ACTION Robi_PallWait_action:
Robot01.PosNo:=POS_FEED_PAL_WAIT;
	Robot01.PosOffset:=gRobotOffset;
	Robot01.Override:=MP.ST00.Override;
	Robot01.SetToolOn:=FALSE;
	Robot01.SetToolOff:=TRUE;
	Robot01.ExecuteMove:=TRUE;
END_ACTION

ACTION Release_Nest_2_action:
ST00_71_K2.SetSignalHigh:=TRUE; (* Schnittstelle Bedrucken Tinte Abholposition frei *)
END_ACTION

ACTION ST08_Pallett_5_entry:
ProcessMessage01:='';
END_ACTION

ACTION ST08_Pallett_5_action:
ProcessMessage01:='1IM7';(*warte Pallette*)
END_ACTION

ACTION ST08_Pallett_5_exit:
ST08_Process.Start:=FALSE;
ProcessMessage01:='';
END_ACTION

ACTION Robot01_PosPal_5_entry:
IF 	PosIdx<TD.PartsInRoboGripper THEN
	PosIdx:=TD.PartsInRoboGripper;
END_IF

(*für das ausschleusen der Testteile mit einem Blister*)
IF	(gTakeTestParts OR gTakeTestPartsAuto) AND
	PosIdx <= MP.ST03.NoOfTestParts THEN
	CTR:=PosIdx;
END_IF
END_ACTION

ACTION Robot01_PosPal_5_action:
Robot01.PosNo:=POS_FEED_PAL_WAIT + (PosIdx/TD.PartsInRoboGripper);
Robot01.PosOffset:=gRobotOffset;
Robot01.Override:=MP.ST00.Override;
Robot01.SetToolOn:=TRUE;
Robot01.SetToolOff:=FALSE;
Robot01.ExecuteMove:=TRUE;
END_ACTION

ACTION Robot01_PosPal_5_exit:
gRob01GripState:=PART_NO;
PosIdx:=PosIdx+ TD.PartsInRoboGripper;
gPartsInserted:=gPartsInserted+ TD.PartsInRoboGripper;
gPartsTest:=gPartsTest+ TD.PartsInRoboGripper;
END_ACTION

ACTION Reset_Test2_action:
(*für das ausschleusen der Testteile mit einem Blister*)
IF	(gTakeTestParts OR gTakeTestPartsAuto) AND
	CTR>= MP.ST03.NoOfTestParts THEN
	ST08_Palletizing.TestpartMoveOut:=TRUE;
	CTR:=0;
	gTakeTestParts:=FALSE;
	gTakeTestPartsAuto:=FALSE;
	TestPartsRemove := TRUE;
END_IF
END_ACTION

ACTION Release_Nest_21_action:
ST00_71_K2.SetSignalHigh:=TRUE; (* Schnittstelle Bedrucken Tinte Abholposition frei *)
END_ACTION

ACTION ST08_Pallett_51_action:
IF ST08_Process.State=STATE_WAIT THEN
	ST08_Process.Start:=TRUE;
END_IF
END_ACTION

ACTION Robot01_Pos51_action:
Robot01.PosNo:=POS_NOK;
Robot01.PosOffset:=gRobotOffset;
Robot01.Override:=MP.ST00.Override;
Robot01.SetToolOn:=TRUE;
Robot01.SetToolOff:=FALSE;
Robot01.ExecuteMove:=TRUE;
END_ACTION

ACTION Robot01_TestPos__entry:
CTR:=CTR+1;
END_ACTION

ACTION Robot01_TestPos__action:
Robot01.PosNo:=POS_TEST_PARTS ;
Robot01.PosOffset:=gRobotOffset;
Robot01.Override:=MP.ST00.Override;
Robot01.SetToolOn:=TRUE;
Robot01.SetToolOff:=FALSE;
Robot01.ExecuteMove:=TRUE;
END_ACTION

ACTION Robot01_TestPos__exit:
gRob01GripState:=PART_NO;
END_ACTION

ACTION Reset_Test__action:
IF CTR>=MP.ST03.NoOfTestParts THEN
	CTR:=0;
	gTakeTestParts:=FALSE;
	gTakeTestPartsAuto:=FALSE;
	TestPartsRemove:=TRUE;
END_IF
END_ACTION

ACTION Robot01_POS_PARK_12_action:
Robot01.PosNo:=POS_PARK;
Robot01.PosOffset:=gRobotOffset;
Robot01.Override:=MP.ST00.Override;
Robot01.SetToolOn:=FALSE;
Robot01.SetToolOff:=FALSE;
Robot01.ExecuteMove:=TRUE;
END_ACTION

ACTION Close_Stopper____________action:
ST03_422_Y64_6.MoveInit:=TRUE;
END_ACTION

ACTION Open_Seperator__________action:
ST03_422_Y64_5.MoveInit:=TRUE;	(* Förderband  Stopper Vereinzler AST/GST *)
END_ACTION

ACTION Wait__for_Part_____entry:
ProcessMessage01:='';
Delay.IN:=FALSE;
Delay();
END_ACTION

ACTION Wait__for_Part_____action:
ProcessMessage01:='1IM6';(*warte auf Teil in Vereinzelung*)
Delay.IN:= ST03_421_B63_7.BitInToCheck; 			 (* Schnittstelle Iso auf Übergabeposition *)
Delay.PT:=T#500ms;
Delay();
END_ACTION

ACTION Wait__for_Part_____exit:
ProcessMessage01:='';
END_ACTION

ACTION Close__seperator__action:
ST03_422_Y64_5.MoveWork:=TRUE;
END_ACTION

ACTION Open__Stopper___action:
ST03_422_Y64_6.MoveWork:=TRUE;
END_ACTION

ACTION Wait_for__Part___entry:
ProcessMessage01:='';
Delay.IN:=FALSE;
Delay();
END_ACTION

ACTION Wait_for__Part___action:
ProcessMessage01:='1IM10';(*warte auf Teil in Abholpositon*)
Delay.IN:=ST03_422_B64_4.BitInToCheck; 		 (* Teil auf Abholposition Roboter *)
Delay.PT:=T#500ms;
Delay();
END_ACTION

ACTION Wait_for__Part___exit:
ProcessMessage01:='';
END_ACTION

ACTION Close_Stopper_2___________action:
ST03_422_Y64_6.MoveInit:=TRUE;
END_ACTION

ACTION Open_Seperator_2_________action:
ST03_422_Y64_5.MoveInit:=TRUE;	(* Förderband  Stopper Vereinzler AST/GST *)
END_ACTION

ACTION Close_Stopper__action:
ST08_412_Y55_2.MoveWork:=TRUE;
END_ACTION

ACTION Open_seperator__action:
ST08_412_Y55_0.MoveInit:=TRUE;
END_ACTION

ACTION Wait_for_Part__entry:
ProcessMessage01:='';
Delay.IN:=FALSE;
Delay();
END_ACTION

ACTION Wait_for_Part__action:
ProcessMessage01:='1IM6';(*warte auf Teil in Vereinzelung*)
Delay.IN:=ST08_412_B58_7.BitInToCheck; 		 (* Schnittstelle Iso auf Übergabeposition *)
Delay.PT:=T#50ms;
Delay();
END_ACTION

ACTION Wait_for_Part__exit:
ProcessMessage01:='';
END_ACTION

ACTION Move_Dist_entry:
IstPosHelp:=ST03_51_M1.sPos.ist;
END_ACTION

ACTION Close_seperator__action:
ST08_412_Y55_0.MoveWork:=TRUE;
END_ACTION

ACTION Open_Stopper___action:
ST08_412_Y55_2.MoveInit:=TRUE;
END_ACTION

ACTION Wait_for_Part___entry:
ProcessMessage01:='';
Delay.IN:=FALSE;
Delay();
END_ACTION

ACTION Wait_for_Part___action:
ProcessMessage01:='1IM10';(*warte auf Teil in Abholpositon*)
Delay.IN:=ST08_412_B59_0.BitInToCheck; 		 (* Teil auf Abholposition Roboter *)
Delay.PT:=T#500ms;
Delay();
END_ACTION

ACTION Wait_for_Part___exit:
ProcessMessage01:='';
END_ACTION

ACTION Close_Stopper_______action:
ST08_412_Y55_2.MoveWork:=TRUE;
END_ACTION

ACTION Open_seperator_______action:
ST08_412_Y55_0.MoveInit:=TRUE;
END_ACTION

ACTION Robot01_Pos35_action:
Robot01.PosNo:=POS_WT_POS2;
Robot01.PosOffset:=gRobotOffset;
Robot01.Override:=MP.ST00.Override;
Robot01.SetToolOn:=FALSE;
Robot01.SetToolOff:=TRUE;
Robot01.ExecuteMove:=TRUE;
END_ACTION

ACTION Robot01_Pos35_exit:
gRob01GripState:=PART_OK;
END_ACTION

ACTION Stopp_Band_91pol_action:
(* Bei 91 poligen Stecker das Band anhalten*)

IF 	gTypeCode=379 THEN
	ST03_51_M1.MotorOn:=FALSE;
	ST03_51_M1.MotorOff :=TRUE;
END_IF
END_ACTION

ACTION Robot01_Pos31_65_action:
Robot01.PosNo:=POS_WT_POS1;
Robot01.PosOffset:=gRobotOffset;
Robot01.Override:=MP.ST00.Override;
Robot01.SetToolOn:=FALSE;
Robot01.SetToolOff:=TRUE;
Robot01.ExecuteMove:=TRUE;
END_ACTION

ACTION Robot01_Pos31_65_exit:
gRob01GripState:=PART_OK;
END_ACTION

ACTION Band_starten_action:
(* Band wieder starten*)

IF 	gTypeCode=379 THEN
	ST03_51_M1.MotorOn:=TRUE;
	ST03_51_M1.MotorOff :=FALSE;
END_IF
END_ACTION

ACTION Robot01__POS_PARK_action:
Robot01.PosNo:=POS_PARK;
Robot01.PosOffset:=gRobotOffset;
Robot01.Override:=MP.ST00.Override;
Robot01.SetToolOn:=FALSE;
Robot01.SetToolOff:=FALSE;
Robot01.ExecuteMove:=TRUE;
END_ACTION

ACTION ST08_Pallett_6_entry:
ProcessMessage01:='';
END_ACTION

ACTION ST08_Pallett_6_action:
ProcessMessage01:='1IM7';(*warte Pallette*)
END_ACTION

ACTION ST08_Pallett_6_exit:
ST08_Process.Start:=FALSE;
ProcessMessage01:='';
END_ACTION

ACTION Robot01_PosPal_65_entry:
IF 	PosIdx<TD.PartsInRoboGripper THEN
	PosIdx:=TD.PartsInRoboGripper;
END_IF

(*für das ausschleusen der Testteile mit einem Blister*)
IF	(gTakeTestParts OR gTakeTestPartsAuto) AND
	PosIdx <= MP.ST03.NoOfTestParts THEN
	CTR:=PosIdx;
END_IF
END_ACTION

ACTION Robot01_PosPal_65_action:
Robot01.PosNo:=POS_FEED_PAL_WAIT + PosIdx;
Robot01.PosOffset:=gRobotOffset;
Robot01.Override:=MP.ST00.Override;
Robot01.SetToolOn:=TRUE;
Robot01.SetToolOff:=FALSE;
Robot01.ExecuteMove:=TRUE;
END_ACTION

ACTION Robot01_PosPal_65_exit:
gRob01GripState:=PART_NO;
PosIdx:=PosIdx+TD.PartsInRoboGripper;
gPartsInserted:=gPartsInserted+TD.PartsInRoboGripper;
gPartsTest:=gPartsTest+ TD.PartsInRoboGripper;
END_ACTION

ACTION Reset_Test3_action:
(*für das ausschleusen der Testteile mit einem Blister*)
IF	(gTakeTestParts OR gTakeTestPartsAuto) AND
	CTR>= MP.ST03.NoOfTestParts THEN
	ST08_Palletizing.TestpartMoveOut:=TRUE;
	CTR:=0;
	gTakeTestParts:=FALSE;
	gTakeTestPartsAuto:=FALSE;
	TestPartsRemove := TRUE;
END_IF
END_ACTION

ACTION ST08_Pallett_8_action:
IF 	ST08_Process.State=STATE_WAIT THEN
	ST08_Process.Start:=TRUE;
END_IF
END_ACTION

ACTION Robot01_POS_PARK_3__action:
Robot01.PosNo:=POS_PARK;
Robot01.PosOffset:=gRobotOffset;
Robot01.Override:=MP.ST00.Override;
Robot01.SetToolOn:=FALSE;
Robot01.SetToolOff:=FALSE;
Robot01.ExecuteMove:=TRUE;
END_ACTION

ACTION Close__seperator_2_action:
ST03_422_Y64_5.MoveWork:=TRUE;
END_ACTION

ACTION Open__Stopper_2__action:
ST03_422_Y64_6.MoveWork:=TRUE;
END_ACTION

ACTION Wait_for_Part____entry:
ProcessMessage01:='';
Delay.IN:=FALSE;
Delay();
END_ACTION

ACTION Wait_for_Part____action:
ProcessMessage01:='1IM10';(*warte auf Teil in Abholpositon*)
Delay.IN:=ST03_422_B64_4.BitInToCheck; 		 (* Teil auf Abholposition Roboter *)
Delay.PT:=T#500ms;
Delay();
END_ACTION

ACTION Wait_for_Part____exit:
ProcessMessage01:='';
END_ACTION

ACTION Close_Stopper_1___________action:
ST03_422_Y64_6.MoveInit:=TRUE;
END_ACTION

ACTION Open_Seperator_1_________action:
ST03_422_Y64_5.MoveInit:=TRUE;	(* Förderband  Stopper Vereinzler AST/GST *)
END_ACTION

ACTION Close_seperator___action:
ST08_412_Y55_0.MoveWork:=TRUE;
END_ACTION

ACTION Open_Stopper____action:
ST08_412_Y55_2.MoveInit:=TRUE;
END_ACTION

ACTION Wait_for_Part_1___entry:
ProcessMessage01:='';
Delay.IN:=FALSE;
Delay();
END_ACTION

ACTION Wait_for_Part_1___action:
ProcessMessage01:='1IM10';(*warte auf Teil in Abholpositon*)
Delay.IN:=ST08_412_B59_0.BitInToCheck; 		 (* Teil auf Abholposition Roboter *)
Delay.PT:=T#500ms;
Delay();
END_ACTION

ACTION Wait_for_Part_1___exit:
ProcessMessage01:='';
END_ACTION

ACTION Close__Stopper_______action:
ST08_412_Y55_2.MoveWork:=TRUE;
END_ACTION

ACTION Open_seperator____action:
ST08_412_Y55_0.MoveInit:=TRUE;
END_ACTION

ACTION Robot01_TestPos___entry:
CTR:=CTR+1;
END_ACTION

ACTION Robot01_TestPos___action:
Robot01.PosNo:=POS_TEST_PARTS ;
Robot01.PosOffset:=gRobotOffset;
Robot01.Override:=MP.ST00.Override;
Robot01.SetToolOn:=TRUE;
Robot01.SetToolOff:=FALSE;
Robot01.ExecuteMove:=TRUE;
END_ACTION

ACTION Robot01_TestPos___exit:
gRob01GripState:=PART_NO;
END_ACTION

ACTION Reset_Test___action:
IF CTR>=MP.ST03.NoOfTestParts
THEN
	CTR:=0;
	gTakeTestParts:=FALSE;
	gTakeTestPartsAuto:=FALSE;
END_IF
END_ACTION

ACTION Robot01_POS_PARK_3_action:
Robot01.PosNo:=POS_PARK;
Robot01.PosOffset:=gRobotOffset;
Robot01.Override:=MP.ST00.Override;
Robot01.SetToolOn:=FALSE;
Robot01.SetToolOff:=FALSE;
Robot01.ExecuteMove:=TRUE;
END_ACTION

ACTION ST02_Main_Print_exit:
ST02_Main.Start:=FALSE;
SFCRun:=FALSE;
END_ACTION

ACTION Robot01_Pos21_action:
Robot01.PosNo:=POS_RT;
Robot01.PosOffset:=gRobotOffset;
Robot01.Override:=MP.ST00.Override;
Robot01.SetToolOn:=FALSE;
Robot01.SetToolOff:=TRUE;
Robot01.ExecuteMove:=TRUE;
END_ACTION

ACTION Robot01_Pos21_exit:
IF	MP.ST02.TableData[1].ProcessData.	Result =11 THEN
	gRob01GripState:= PART_OK;
ELSE
	gRob01GripState:=PART_NOK;
END_IF
END_ACTION

ACTION set_PartState_exit:
Result_help:=MP.ST02.TableData[1].ProcessData.Result;
MP.ST02.TableData[1].ProcessData.Part:= FALSE; 		 (* Schnittstelle Tampondrucker Nest 1 leer *)
MP.ST02.TableData[1].ProcessData.Result:=0;	(*   0 = Teil noch nicht bearbeitet *)
											(*   1 =  Oberseite OK*)
											(*  11 = Oberseite und Unterseite OK*)
											(*  99 = Teil ist NOK	*)
END_ACTION

ACTION Robo01_PosNOK_action:
Robot01.PosNo:=POS_NOK;
Robot01.PosOffset:=gRobotOffset;
Robot01.Override:=MP.ST00.Override;
Robot01.SetToolOn:=TRUE;
Robot01.SetToolOff:=FALSE;
Robot01.ExecuteMove:=TRUE;
END_ACTION

ACTION Robo01_PosNOK_exit:
gRob01GripState:=PART_NO;
IF	Result_help =11 THEN
	PutIdx:=PutIdx+1;
	i32_first_parts :=i32_first_parts+1;
END_IF
END_ACTION

ACTION ST08_Pallett_33_entry:
ProcessMessage01:='';
END_ACTION

ACTION ST08_Pallett_33_action:
ProcessMessage01:='1IM7';(*warte Pallette*)
END_ACTION

ACTION ST08_Pallett_33_exit:
ST08_Process.Start:=FALSE;
ProcessMessage01:='';
END_ACTION

ACTION Robot01_POS_PARK_action:
Robot01.PosNo:=POS_PARK;
Robot01.PosOffset:=gRobotOffset;
Robot01.Override:=MP.ST00.Override;
Robot01.SetToolOn:=FALSE;
Robot01.SetToolOff:=FALSE;
Robot01.ExecuteMove:=TRUE;
END_ACTION

ACTION ST08_Pallett_3_entry:
ProcessMessage01:='';
END_ACTION

ACTION ST08_Pallett_3_action:
ProcessMessage01:='1IM7';(*warte Pallette*)
END_ACTION

ACTION ST08_Pallett_3_exit:
ST08_Process.Start:=FALSE;
ProcessMessage01:='';
END_ACTION

ACTION Robot01_PosPal_entry:
IF 	PosIdx<TD.PartsInRoboGripper THEN
	PosIdx:=TD.PartsInRoboGripper;
END_IF

(*für das ausschleusen der Testteile mit einem Blister*)
IF	(gTakeTestParts OR gTakeTestPartsAuto) AND
	PosIdx <= MP.ST03.NoOfTestParts THEN
	CTR:=PosIdx;
END_IF
END_ACTION

ACTION Robot01_PosPal_action:
Robot01.PosNo:=POS_FEED_PAL_WAIT + (PosIdx/TD.PartsInRoboGripper);
Robot01.PosOffset:=gRobotOffset;
Robot01.Override:=MP.ST00.Override;
Robot01.SetToolOn:=TRUE;
Robot01.SetToolOff:=FALSE;
Robot01.ExecuteMove:=TRUE;
END_ACTION

ACTION Robot01_PosPal_exit:
gRob01GripState:=PART_NO;
PosIdx:=PosIdx+TD.PartsInRoboGripper;
gPartsInserted:=gPartsInserted+TD.PartsInRoboGripper;
gPartsTest:=gPartsTest+TD.PartsInRoboGripper;
END_ACTION

ACTION Reset_Test1_action:
(*für das ausschleusen der Testteile mit einem Blister*)
IF	(gTakeTestParts OR gTakeTestPartsAuto) AND
	CTR>= MP.ST03.NoOfTestParts THEN
	ST08_Palletizing.TestpartMoveOut:=TRUE;
	CTR:=0;
	gTakeTestParts:=FALSE;
	gTakeTestPartsAuto:=FALSE;
	TestPartsRemove := TRUE;
END_IF
END_ACTION

ACTION ST08_Pallett_action:
IF 	ST08_Process.State=STATE_WAIT THEN
	ST08_Process.Start:=TRUE;
END_IF
END_ACTION

ACTION RemoveTestParts_entry:
MessageHandler.ClearMessageLines(sVisu:=Visu.Message);
END_ACTION

ACTION RemoveTestParts_action:
IF  ST03_8_75_B13_5.SignalIn THEN		(*voll/belegt keine Prüfmittel mehr  *)
	MessageHandler.Msg.ID:='PM116';
ELSIF ST03_8_75_B13_6.SignalIn THEN	(* belegt mit 6 Prüfmittel  *)
	MessageHandler.Msg.ID:='PM117';
END_IF

MessageHandler.Msg.Name:='Prüfteile entnehmen';
MessageHandler.Msg.Text:='Kontrolle ob die Rutsche leer ist.';
MessageHandler.Msg.Color:=Color.red;
MessageHandler.Msg.Station:=1;


MessageHandler(
	Prio:=2, 							(*1=highest, .. , 4=lowest*)
	Btn1Addr:=ADR(MsgOk),			(*Address of Button1 , if Zero then Button is unvisible*)
	Btn2Addr:=0,						(*Address of Button2 , if Zero then Button is unvisible*)
	sVisu:=Visu.Message);
END_ACTION

ACTION RemoveTestParts_exit:
MsgOk:=FALSE;
MsgCancel:=FALSE;
END_ACTION

ACTION Robot01_TestPos_entry:
CTR:=CTR+1;
CTR2:=CTR2+1;
END_ACTION

ACTION Robot01_TestPos_action:
Robot01.PosNo:=POS_TEST_PARTS;
Robot01.PosOffset:=gRobotOffset;
Robot01.Override:=MP.ST00.Override;
Robot01.SetToolOn:=TRUE;
Robot01.SetToolOff:=FALSE;
Robot01.ExecuteMove:=TRUE;
END_ACTION

ACTION Robot01_TestPos_exit:
gRob01GripState:=PART_NO;
i32_first_parts :=i32_first_parts+1;
END_ACTION

ACTION Step140_action:
IF ST02_Main.State=STATE_WAIT THEN
	ST02_Main.Start:=TRUE;
END_IF
END_ACTION

ACTION Robot01_Pos21____action:
Robot01.PosNo:=POS_RT;
Robot01.PosOffset:=gRobotOffset;
Robot01.Override:=MP.ST00.Override;
Robot01.SetToolOn:=FALSE;
Robot01.SetToolOff:=TRUE;
Robot01.ExecuteMove:=TRUE;
END_ACTION

ACTION Robot01_Pos21____exit:
IF	MP.ST02.TableData[1].ProcessData.	Result =11 THEN
	gRob01GripState:= PART_OK;
ELSE
	gRob01GripState:=PART_NOK;
END_IF
END_ACTION

ACTION Reset_Test_action:
IF NOT MP.ST02.DummyPruefung_93pol AND
 CTR=MP.ST03.NoOfTestParts
THEN
	CTR:=0;
	gTakeTestParts:=FALSE;
	gTakeTestPartsAuto:=FALSE;
	TestPartsRemove:=TRUE;
ELSIF
	 CTR2 = MP.ST02.NoOfDummys THEN
	CTR2:=0;
	MP.ST02.DummyPruefung_93pol:= FALSE;
END_IF
END_ACTION

ACTION Robot01_POS32__action:
Robot01.PosNo:=POS_WT_POS1_WAIT;
Robot01.PosOffset:=gRobotOffset;
Robot01.Override:=MP.ST00.Override;
Robot01.SetToolOn:=FALSE;
Robot01.SetToolOff:=FALSE;
Robot01.ExecuteMove:=TRUE;
END_ACTION

ACTION Robot01_Pos31_action:
Robot01.PosNo:=POS_WT_POS1;
Robot01.PosOffset:=gRobotOffset;
Robot01.Override:=MP.ST00.Override;
Robot01.SetToolOn:=FALSE;
Robot01.SetToolOff:=TRUE;
Robot01.ExecuteMove:=TRUE;
END_ACTION

ACTION Robot01_Pos31_exit:
gRob01GripState:=PART_NEW;
END_ACTION

ACTION Robot01_POS22_action:
Robot01.PosNo:=POS_RT_WAIT;
Robot01.PosOffset:=gRobotOffset;
Robot01.Override:=MP.ST00.Override;
Robot01.SetToolOn:=FALSE;
Robot01.SetToolOff:=FALSE;
Robot01.ExecuteMove:=TRUE;
END_ACTION

ACTION Handshake_entry:
Nest_Empty:=TRUE;
END_ACTION

ACTION Handshake_exit:
Nest_Empty:=FALSE;
END_ACTION

ACTION Robot01_Pos21__action:
Robot01.PosNo:=POS_RT;
Robot01.PosOffset:=gRobotOffset;
Robot01.Override:=MP.ST00.Override;
Robot01.SetToolOn:=TRUE;
Robot01.SetToolOff:=FALSE;
Robot01.ExecuteMove:=TRUE;
END_ACTION

ACTION Robot01_Pos21__exit:
gRob01GripState:=PART_NO;
gRTState[1]:=PART_NEW;
END_ACTION

ACTION set_PartState__exit:
MP.ST02.TableData[1].ProcessData.Part:= TRUE; 		 (* Schnittstelle Tampondrucker Nest 1 leer *)
MP.ST02.TableData[1].ProcessData.Result:=0;	(*   0 = Teil noch nicht bearbeitet *)
											(*   1 =  Oberseite OK*)
											(*  11 = Oberseite und Unterseite OK*)
											(*  99 = Teil ist NOK	*)
END_ACTION

ACTION Robot01_POS23__action:
Robot01.PosNo:=23;
Robot01.PosOffset:=gRobotOffset;
Robot01.Override:=MP.ST00.Override;
Robot01.SetToolOn:=FALSE;
Robot01.SetToolOff:=FALSE;
Robot01.ExecuteMove:=TRUE;
END_ACTION

ACTION ST02_Main_Print__action:
IF 	ST02_Main.State=STATE_WAIT THEN
	ST02_Main.Start:=TRUE;
END_IF
END_ACTION

ACTION ST02_Main_Print__exit:
ST02_Main.Start:=FALSE;
END_ACTION

ACTION Wait_Printer_finish__entry:
ProcessMessage01:='';
Delay.IN:=FALSE;
Delay();
END_ACTION

ACTION Wait_Printer_finish__action:
ProcessMessage01:='1IM23';(*warte auf Druck fertig*)
Delay.IN:=TRUE;

IF MP.ST00.Override >0 AND gTipImp THEN
	DElay.PT:=t#4000s / MP.ST00.Override;
ELSE
	DElay.PT:=t#1h;
END_IF

Delay();
END_ACTION

ACTION Wait_Printer_finish__exit:
ProcessMessage01:='';
END_ACTION

ACTION Open_Stopper3_action:
ST00_74_Y2_4.MoveWork:=TRUE;
END_ACTION

ACTION Msg_Error___entry:
MessageHandler.ClearMessageLines(sVisu:=Visu.Message);
END_ACTION

ACTION Msg_Error___action:
MessageHandler.Msg.ID:='PM115';
MessageHandler.Msg.Name:='Drucker';
MessageHandler.Msg.Text:='Kein Betriebsbereit vom Drucker ';
MessageHandler.Msg.Color:=Color.Red;
MessageHandler.Msg.Station:=1;


MessageHandler(
	Prio:=2, 									(*1=highest, .. , 4=lowest*)
	Btn1Addr:=ADR(MsgOk),			(*Address of Button1 , if Zero then Button is unvisible*)
	Btn2Addr:=0,	(*Address of Button2 , if Zero then Button is unvisible*)
	sVisu:=Visu.Message);
END_ACTION

ACTION Msg_Error___exit:
MessageHandler.ClearMessageLines(sVisu:=Visu.Message);
MsgOk:=FALSE;
END_ACTION

ACTION Close_Stopper44_action:
ST00_74_Y2_4.MoveInit:=TRUE;
END_ACTION

ACTION Fertig_entry:
gRTState[1]:=gRTState[2];
gRTState[2]:=PART_OK;
END_ACTION

ACTION Robot01_Pos1__1__action:
Robot01.PosNo:=POS_PARK;
Robot01.PosOffset:=gRobotOffset;
Robot01.Override:=MP.ST00.Override;
(*Robot01.SetToolOn:=TRUE;
Robot01.SetToolOff:=FALSE;*)
Robot01.ExecuteMove:=TRUE;
END_ACTION

ACTION Robot01_Pos1__1__exit:
ST08_Process.Start:=FALSE;
END_ACTION

ACTION SeqEnd_action:
SFCTime:=TIME_TO_DINT(TIME()-SFCTimeStart);
State:=STATE_WAIT;
END_ACTION

TRANSITION CheckPartsInRoboGripper:
TD.PartsInRoboGripper > 0 (*Diffision durch 0 verhindern*)
END_TRANSITION

TRANSITION StateOk:
ST08_Process.State=STATE_OK
END_TRANSITION

TRANSITION No_Part:
gRob01GripState=PART_NO
END_TRANSITION

TRANSITION Part_OK_:
gRob01GripState = PART_OK AND
((NOT MP.ST08.TrayAushebenMotor AND ST08_406_B54_4.ValveSensor) OR	(* Ausheber Trays Entnahmepos. Isok. STN8 AST *)
(MP.ST08.TrayAushebenMotor AND ABS(ST08_190_M1.sPos.ist - TD.PosTrayAusheben[2].Pos) < 0.5)) (*1=unten, 2=oben, *)
END_TRANSITION

TRANSITION StateOK:
Robot01.State=STATE_OK
END_TRANSITION

TRANSITION StateOk:
ST08_Process.State=STATE_OK
END_TRANSITION

TRANSITION #StateOK:
Robot01.State=STATE_OK

AND gTipImp
END_TRANSITION

TRANSITION Part_New:
gRob01GripState=PART_NEW AND
gTypeCode=312
END_TRANSITION

TRANSITION Part_Cam:
gRob01GripState=PART_CAM (*Teil im Greifer ohne Kameraprüfung*)
END_TRANSITION

TRANSITION RT_Nest_empty:
     (ST02_DT_65B11.BitInToCheck      (* Tampondrucker Nest 1 leer *)
 	 AND ST02_DT_62_B91.ValveSensor )	     (* Tampondrucker Nest 1 in Abholposition *)

OR
	   (ST02_DT_65B21.BitInToCheck  		 (* Tampondrucker Nest 2 leer *)
  AND ST02_DT_62_B81.ValveSensor )     (* Tampondrucker Nest 2 in Abholposition *)
END_TRANSITION

TRANSITION #StateOK:
Robot01.State=STATE_OK

AND gTipImp
END_TRANSITION

TRANSITION all_other:
(gTypeCode<>4991 AND	(*102 pol*)
 gTypeCode<>312) 		(*93 pol*)
END_TRANSITION

TRANSITION 93-102polig:
(gTypeCode=4991 OR 	(*102 pol*)
 gTypeCode=312) 	(*93 pol*)

AND
(ST02_DT_62_B81.ValveSensor OR	(* Tampondrucker Nest 1 in Abholposition *)
 ST02_DT_62_B91.ValveSensor )		(* Tampondrucker Nest 2 in Abholposition *)
END_TRANSITION

TRANSITION Printer_off:
NOT ST02_DT_62_B81.ValveSensor	 AND	     (* Tampondrucker Nest 1 in Abholposition *)
NOT ST02_DT_62_B91.ValveSensor 		     (* Tampondrucker Nest 2 in Abholposition *)
END_TRANSITION

TRANSITION StateOk:
ST00_74_Y2_4.State=STATE_OK
END_TRANSITION

TRANSITION StateOk:
ST00_74_Y2_5.State=STATE_OK
END_TRANSITION

TRANSITION Finish:
	ST00_72_X1_8.BitInToCheck (* Schnittstelle Tampondrucker Druck abgeschlossen *)
END_TRANSITION

TRANSITION StateOk:
ST00_74_Y2_4.State=STATE_OK
END_TRANSITION

TRANSITION 93_102polig:
(*mit Tampondrucker*)
gTypeCode=4991 OR 	(*102 pol*)
gTypeCode=312		(*93 pol*)
END_TRANSITION

TRANSITION 268pol:
gTypeCode=5841 (* AND 	(*268 pol*)
ST03_8_100_A1.Activated*)
END_TRANSITION

TRANSITION CamDone:
(gRob01GripState=PART_OK OR
gRob01GripState=PART_NOK) AND
ST03_268pol_Zufuehrung.State=STATE_WAIT
END_TRANSITION

TRANSITION 102pol_neu:
gTypeCode=4993 (*  AND 	(*102 pol neu*)
ST03_8_100_A1.Activated*)
END_TRANSITION

TRANSITION CamDone:
(gRob01GripState=PART_OK OR
gRob01GripState=PART_NOK) AND
ST03_102pol_neu_Zufuehrung.State=STATE_WAIT
END_TRANSITION

TRANSITION all_other_polig:
(*Tampondrucker*)
(gTypeCode<>4991 AND(*102 pol*)
gTypeCode<>312) AND	(*93 pol*)

(*alte Rüstsätze*)
gTypeCode<>360  AND	(*74pol*)
(*gTypeCode<>379  AND*)	(*91pol*)
gTypeCode<>4992 AND	(*35pol*)
gTypeCode<>489		(*168pol*)
END_TRANSITION

TRANSITION Part_Ready_Pick:
Delay.Q
END_TRANSITION

TRANSITION AutoStop:
		ModeSelect.Mode=MODE_AUTO_STOP
OR	ModeSelect.Mode=MODE_STEP_STOP
END_TRANSITION

TRANSITION POS_1:
ST03_Init_AbholPos.RoboPos31
END_TRANSITION

TRANSITION POS_2:
ST03_Init_AbholPos.RoboPos35
END_TRANSITION

TRANSITION #StateOK:
Robot01.State=STATE_OK

AND gTipImp
END_TRANSITION

TRANSITION #StateOK:
Robot01.State=STATE_OK

AND gTipImp
END_TRANSITION

TRANSITION Yes:
(
gTakeTestParts OR
gTakeTestPartsAuto)
AND
NOT TD.TestpartBilister AND
gRob01GripState = PART_OK AND
NOT ST03_8_75_B13_5.BitInToCheck
END_TRANSITION

TRANSITION i.O.:
gRob01GripState = PART_OK
END_TRANSITION

TRANSITION StateOk:
ST08_Process.State=STATE_OK
OR
gTypeCode=379
END_TRANSITION

TRANSITION StateOk:
Robot01.State=STATE_OK
END_TRANSITION

TRANSITION Pal_OK:
ST08_Process.Pal_Ready AND
NOT ST08_Palletizing.TestpartMoveOut AND
((NOT MP.ST08.TrayAushebenMotor AND ST08_406_B54_4.ValveSensor) OR	(* Ausheber Trays Entnahmepos. Isok. STN8 AST *)
(MP.ST08.TrayAushebenMotor AND ABS(ST08_190_M1.sPos.ist - TD.PosTrayAusheben[2].Pos) < 0.5)) (*1=unten, 2=oben, *)
END_TRANSITION

TRANSITION allOther:
gTypeCode<>379 AND	(*91 pol*)
gTypeCode<>4993		(*102pol neu*)
END_TRANSITION

TRANSITION StateOk:
Robot01.State=STATE_OK
END_TRANSITION

TRANSITION OK:
ST00_71_K2.State=State_OK
END_TRANSITION

TRANSITION StateOk:
ST08_Process.State=STATE_OK OR
ST08_Process.State=STATE_Wait
END_TRANSITION

TRANSITION Pal_OK:
ST08_Process.Pal_Ready AND
NOT ST08_Palletizing.TestpartMoveOut AND
((NOT MP.ST08.TrayAushebenMotor AND ST08_406_B54_4.ValveSensor) OR	(* Ausheber Trays Entnahmepos. Isok. STN8 AST *)
(MP.ST08.TrayAushebenMotor AND ABS(ST08_190_M1.sPos.ist - TD.PosTrayAusheben[2].Pos) < 0.5)) (*1=unten, 2=oben, *)
END_TRANSITION

TRANSITION StateOK:
Robot01.State=STATE_OK
END_TRANSITION

TRANSITION OK:
ST00_71_K2.State=State_OK
END_TRANSITION

TRANSITION StateRun:
ST08_Process.State=STATE_Run OR
gRunEmpty
END_TRANSITION

TRANSITION n.i.O:
gRob01GripState = PART_NOK
END_TRANSITION

TRANSITION #StateOK:
Robot01.State=STATE_OK

AND gTipImp
END_TRANSITION

TRANSITION StateOK:
Robot01.State=STATE_OK
END_TRANSITION

TRANSITION empty:
NOT ST03_8_75_B13_5.BitInToCheck
END_TRANSITION

TRANSITION #StateOK:
Robot01.State=STATE_OK

AND gTipImp
END_TRANSITION

TRANSITION T9_74_168_35polig:
(*alte Rüstsätze*)
gTypeCode=360 OR	(*74pol*)
(*gTypeCode=379 OR*)	(*91pol*)
gTypeCode=4992 OR	(*35pol*)
gTypeCode=489		(*168pol*)
END_TRANSITION

TRANSITION all_other:
NOT MP.ST03.SGM_3621
END_TRANSITION

TRANSITION SGM_3621:
MP.ST03.SGM_3621
END_TRANSITION

TRANSITION leer:
NOT ST03_422_B64_4.BitInToCheck 		 (* Teil auf Abholpos *)
END_TRANSITION

TRANSITION StateOK:
ST03_422_Y64_6.State=STATE_OK
END_TRANSITION

TRANSITION StateOK:
ST03_422_Y64_5.State=STATE_OK
END_TRANSITION

TRANSITION Part_Ready_Print:
Delay.Q
END_TRANSITION

TRANSITION AutoStop:
		ModeSelect.Mode=MODE_AUTO_STOP
OR	ModeSelect.Mode=MODE_STEP_STOP
END_TRANSITION

TRANSITION StateOk:
ST03_422_Y64_5.State=STATE_OK
END_TRANSITION

TRANSITION StateOk:
ST03_422_Y64_6.State=STATE_OK
END_TRANSITION

TRANSITION Part_Ready_Roboter:
Delay.Q
END_TRANSITION

TRANSITION AutoStop:
		ModeSelect.Mode=MODE_AUTO_STOP
OR	ModeSelect.Mode=MODE_STEP_STOP
END_TRANSITION

TRANSITION StateOK:
ST03_422_Y64_6.State=STATE_OK
END_TRANSITION

TRANSITION StateOK:
ST03_422_Y64_5.State=STATE_OK
END_TRANSITION

TRANSITION Abholpos_leer:
NOT ST08_412_B59_0.BitInToCheck 		 (* Teil auf Abholpos *)
END_TRANSITION

TRANSITION StateOk:
ST08_412_Y55_2.State=STATE_OK
END_TRANSITION

TRANSITION StateOk:
ST08_412_Y55_0.State=STATE_OK
END_TRANSITION

TRANSITION Part_Ready_Print:
Delay.Q
END_TRANSITION

TRANSITION AutoStop:
		ModeSelect.Mode=MODE_AUTO_STOP
OR	ModeSelect.Mode=MODE_STEP_STOP
END_TRANSITION

TRANSITION Wait_Pos:
(ST03_51_M1.sPos.ist >
IstPosHelp +TD.DistIso AND MP.ST03.BandMoveP)

OR
(ST03_51_M1.sPos.ist <
IstPosHelp + TD.DistIso AND NOT MP.ST03.BandMoveP)
END_TRANSITION

TRANSITION StateOk:
ST08_412_Y55_0.State=STATE_OK
END_TRANSITION

TRANSITION StateOk:
ST08_412_Y55_2.State=STATE_OK
END_TRANSITION

TRANSITION Part_Ready_Roboter:
Delay.Q
END_TRANSITION

TRANSITION AutoStop:
		ModeSelect.Mode=MODE_AUTO_STOP
OR	ModeSelect.Mode=MODE_STEP_STOP
END_TRANSITION

TRANSITION StateOk:
ST08_412_Y55_2.State=STATE_OK
END_TRANSITION

TRANSITION StateOk:
ST08_412_Y55_0.State=STATE_OK
END_TRANSITION

TRANSITION not_35pol_or_links:
ST03_Init_AbholPos.RoboPos31
END_TRANSITION

TRANSITION 35pol_rechts:
ST03_Init_AbholPos.RoboPos35
END_TRANSITION

TRANSITION #StateOK:
Robot01.State=STATE_OK

AND gTipImp
END_TRANSITION

TRANSITION #StateOK:
Robot01.State=STATE_OK

AND gTipImp
END_TRANSITION

TRANSITION #StateOK:
Robot01.State=STATE_OK

AND gTipImp
END_TRANSITION

TRANSITION Yes:
(gTakeTestParts OR
gTakeTestPartsAuto)
AND
NOT TD.TestpartBilister
AND
NOT ST03_8_75_B13_5.BitInToCheck
END_TRANSITION

TRANSITION No:
gRob01GripState = PART_OK
END_TRANSITION

TRANSITION StateOk:
ST08_Process.State=STATE_OK
END_TRANSITION

TRANSITION StateWait:
ST08_Process.State=STATE_Wait
END_TRANSITION

TRANSITION Pal_OK:
ST08_Process.Pal_Ready
END_TRANSITION

TRANSITION AutoStop:
		ModeSelect.Mode=MODE_AUTO_STOP
OR	ModeSelect.Mode=MODE_STEP_STOP
END_TRANSITION

TRANSITION StateOK:
Robot01.State=STATE_OK
END_TRANSITION

TRANSITION StateRun:
ST08_Process.State=STATE_Run
END_TRANSITION

TRANSITION #StateOK:
Robot01.State=STATE_OK

AND gTipImp
END_TRANSITION

TRANSITION Iso_an_Vereinzler:
ST08_412_B58_7.BitInToCheck 		 (* Schnittstelle Iso auf Übergabeposition *)
OR
 ST03_421_B63_7.BitInToCheck (* für SGM 3621 *)
END_TRANSITION

TRANSITION Trans151:
Robot01.ActualArea <> 4
END_TRANSITION

TRANSITION all_other:
NOT MP.ST03.SGM_3621
END_TRANSITION

TRANSITION SGM_3621:
MP.ST03.SGM_3621
END_TRANSITION

TRANSITION StateOk:
ST03_422_Y64_5.State=STATE_OK
END_TRANSITION

TRANSITION StateOk:
ST03_422_Y64_6.State=STATE_OK
END_TRANSITION

TRANSITION Part_Ready_Roboter:
Delay.Q
END_TRANSITION

TRANSITION StateOK:
ST03_422_Y64_6.State=STATE_OK
END_TRANSITION

TRANSITION StateOK:
ST03_422_Y64_5.State=STATE_OK
END_TRANSITION

TRANSITION StateOk:
ST08_412_Y55_0.State=STATE_OK
END_TRANSITION

TRANSITION StateOk:
ST08_412_Y55_2.State=STATE_OK
END_TRANSITION

TRANSITION Part_Ready_Roboter:
Delay.Q
END_TRANSITION

TRANSITION StateOk:
ST08_412_Y55_2.State=STATE_OK
END_TRANSITION

TRANSITION StateOk:
ST08_412_Y55_0.State=STATE_OK
END_TRANSITION

TRANSITION StateOK:
Robot01.State=STATE_OK
END_TRANSITION

TRANSITION #StateOK:
Robot01.State=STATE_OK

AND gTipImp
END_TRANSITION

TRANSITION Part_Ready_Print:
(NOT ST02_DT_65B11.BitInToCheck AND	(* Tampondrucker Nest 1 leer *)
ST02_DT_61_B51.ValveSensor AND			(* Schwenkarm 1 90 Grad*)
ST02_DT_62_B91.ValveSensor)				(* Tampondrucker Nest 1 in Abholposition 180°*)
OR
(NOT ST02_DT_65B21.BitInToCheck AND	(* Tampondrucker Nest 2 leer *)
ST02_DT_61_B21.ValveSensor AND			(* Schwenkarm 2 90 Grad*)
ST02_DT_62_B81.ValveSensor)			 	(* Tampondrucker Nest 2 in Abholposition 0° *)
END_TRANSITION

TRANSITION RT_Nest_empty:
(ST02_DT_65B11.BitInToCheck AND		(* Tampondrucker Nest 1 leer *)
 ST02_DT_62_B91.ValveSensor)		(* Tampondrucker Nest 1 in Abholposition 180°*)
OR
(ST02_DT_65B21.BitInToCheck AND		(* Tampondrucker Nest 2 leer *)
 ST02_DT_62_B81.ValveSensor ) 		(* Tampondrucker Nest 2 in Abholposition 0°*)
END_TRANSITION

TRANSITION Wait_:
ST02_Main.State=State_WAIT
END_TRANSITION

TRANSITION StateOk:
(*SFCRun AND*)
ST02_Main.State=State_WAIT
END_TRANSITION

TRANSITION AutoStop:
(ModeSelect.Mode=MODE_AUTO_STOP OR
ModeSelect.Mode=MODE_STEP_STOP) AND
ST02_Main.State = STATE_WAIT
END_TRANSITION

TRANSITION #StateOK:
Robot01.State=STATE_OK

AND gTipImp
END_TRANSITION

TRANSITION CounterCheck:
MP.ST02.DummyPruefung_93pol OR
 (gRob01GripState = PART_OK
AND
(PutIdx>=AnzahlTeile OR	(*93pol*)
kein_Teil_NOK))
END_TRANSITION

TRANSITION #StateOK:
Robot01.State = STATE_OK

AND gTipImp
END_TRANSITION

TRANSITION Yes:
(gTakeTestParts OR
gTakeTestPartsAuto OR
MP.ST02.DummyPruefung_93pol)
AND
NOT TD.TestpartBilister
END_TRANSITION

TRANSITION No:
NOT MP.ST02.DummyPruefung_93pol
OR
NOT ST03_8_75_B13_5.BitInToCheck
END_TRANSITION

TRANSITION StateOk:
ST08_Process.State=STATE_OK
END_TRANSITION

TRANSITION StateWait:
ST08_Process.State=STATE_Wait
END_TRANSITION

TRANSITION Pal_OK:
ST08_Process.Pal_Ready=TRUE
END_TRANSITION

TRANSITION #StateOK:
Robot01.State=STATE_OK

AND gTipImp
END_TRANSITION

TRANSITION StateOk:
ST08_Process.State=STATE_OK OR ST08_Process.State=STATE_Wait
END_TRANSITION

TRANSITION Pal_OK:
ST08_Process.Pal_Ready=TRUE
END_TRANSITION

TRANSITION StateOK:
Robot01.State=STATE_OK
END_TRANSITION

TRANSITION StateRun:
ST08_Process.State=STATE_Run
END_TRANSITION

TRANSITION Yes:
NOT ST03_8_75_B13_5.SignalIn AND	(*voll/belegt keine Prüfmittel mehr  *)
NOT ST03_8_75_B13_6.SignalIn AND	(* belegt mit 6 Prüfmittel  *)
NOT TestPartsRemove
END_TRANSITION

TRANSITION StateOK:
Robot01.State=STATE_OK
END_TRANSITION

TRANSITION all_other___:
(gTakeTestParts OR
(gTakeTestPartsAuto AND NOT MP.ST02.DummyPruefung_93pol )OR
(MP.ST02.DummyPruefung_93pol AND CTR2 <>5))
AND
NOT TD.TestpartBilister
END_TRANSITION

TRANSITION Last_Dummy:
MP.ST02.DummyPruefung_93pol AND
CTR2 = 5
END_TRANSITION

TRANSITION Part_Ready___:
(NOT ST02_DT_65B11.BitInToCheck AND	(* Tampondrucker Nest 1 leer *)
ST02_DT_61_B51.ValveSensor AND			(* Schwenkarm 1 90 Grad*)
ST02_DT_62_B91.ValveSensor)				(* Tampondrucker Nest 1 in Abholposition 180°*)
OR
(NOT ST02_DT_65B21.BitInToCheck AND	(* Tampondrucker Nest 2 leer *)
ST02_DT_61_B21.ValveSensor AND			(* Schwenkarm 2 90 Grad*)
ST02_DT_62_B81.ValveSensor)			 	(* Tampondrucker Nest 2 in Abholposition 0° *)
END_TRANSITION

TRANSITION #StateOK:
Robot01.State=STATE_OK

AND gTipImp
END_TRANSITION

TRANSITION #StateOK:
Robot01.State=STATE_OK
AND gTipImp
END_TRANSITION

TRANSITION AutoStop:
(ModeSelect.Mode=MODE_AUTO_STOP OR
ModeSelect.Mode=MODE_STEP_STOP) AND
ST02_Main.State = STATE_WAIT
END_TRANSITION

TRANSITION Auto_run:
ModeSelect.Mode<>MODE_AUTO_STOP AND
ModeSelect.Mode<>MODE_STEP_STOP
END_TRANSITION

TRANSITION AutoStop:
ModeSelect.Mode=MODE_AUTO_STOP OR
ModeSelect.Mode=MODE_STEP_STOP
END_TRANSITION

TRANSITION PartReady:
ST03_102pol_Zufuehrung.PartReady
END_TRANSITION

TRANSITION #StateOK:
Robot01.State=STATE_OK

AND gTipImp
END_TRANSITION

TRANSITION #StateOK:
Robot01.State=STATE_OK

AND gTipImp
END_TRANSITION

TRANSITION OK:
NOT ST03_102pol_Zufuehrung.PartReady
END_TRANSITION

TRANSITION AutoStop:
(ModeSelect.Mode=MODE_AUTO_STOP OR
ModeSelect.Mode=MODE_STEP_STOP) AND
ST02_Main.State = STATE_WAIT
END_TRANSITION

TRANSITION Part_Ready_Print:
  ( ST02_DT_65B11.BitInToCheck AND     (* Tampondrucker Nest 1 leer *)
ST02_DT_61_B51.ValveSensor AND		(* Schwenkarm 1 90 Grad*)
ST02_DT_62_B91.ValveSensor)  		(* Tampondrucker Nest 1 in Abholposition *)
OR
  ( ST02_DT_65B21.BitInToCheck AND  	(* Tampondrucker Nest 2 leer *)
ST02_DT_61_B21.ValveSensor AND		(* Schwenkarm 2 90 Grad*)
ST02_DT_62_B81.ValveSensor ) 		(* Tampondrucker Nest 2 in Abholposition *)
END_TRANSITION

TRANSITION AutoStop:
(ModeSelect.Mode=MODE_AUTO_STOP OR
ModeSelect.Mode=MODE_STEP_STOP) AND
ST02_Main.State = STATE_WAIT
END_TRANSITION

TRANSITION #StateOK:
Robot01.State=STATE_OK

AND gTipImp
END_TRANSITION

TRANSITION #StateOK:
Robot01.State=STATE_OK

AND gTipImp
END_TRANSITION

TRANSITION ST02Wait:
ST02_Main.State=STATE_WAIT
END_TRANSITION

TRANSITION turn_done:
ST02_Main.turn_done
END_TRANSITION

TRANSITION IO:
ST02_Main.turn_done
AND
MP.ST02.TableData[1].ProcessData.	Result =11
											(*   0 = Teil noch nicht bearbeitet *)
											(*   1 =  Oberseite OK*)
											(*  11 = Oberseite und Unterseite OK*)
											(*  99 = Teil ist NOK	*)
END_TRANSITION

TRANSITION NIO:
ST02_Main.turn_done
AND

MP.ST02.TableData[1].ProcessData.	Result <>11
AND

((ST02_DT_65B11.BitInToCheck=FALSE AND     (* Tampondrucker Nest 1 leer *)
ST02_DT_62_B91.ValveSensor)  		(* Tampondrucker Nest 1 in Abholposition *)(*180 Grad*)
OR
(ST02_DT_65B21.BitInToCheck=FALSE AND  	(* Tampondrucker Nest 2 leer *)
ST02_DT_62_B81.ValveSensor )) 		(* Tampondrucker Nest 2 in Abholposition *)(*0 Grad*)
END_TRANSITION

TRANSITION emty:
(ST02_DT_62_B91.ValveSensor AND	(* Tampondrucker Nest 1 in Abholposition *) (*180 Grad*)
 ST02_DT_65B11.BitInToCheck)     		(* Tampondrucker Nest 1 leer *)

OR
(ST02_DT_62_B81.ValveSensor AND 	(* Tampondrucker Nest 2 in Abholposition *)(*0 Grad*)
 ST02_DT_65B21.BitInToCheck) 		 (* Tampondrucker Nest 2 leer *)
END_TRANSITION

TRANSITION Time_out:
Delay.Q
END_TRANSITION

TRANSITION StateOk:
ST00_74_Y2_4.State=STATE_OK
END_TRANSITION

TRANSITION Finish:
 MsgOk
END_TRANSITION

TRANSITION StateOk:
ST00_74_Y2_4.State=STATE_OK
END_TRANSITION

TRANSITION AutoStop:
(ModeSelect.Mode=MODE_AUTO_STOP OR
ModeSelect.Mode=MODE_STEP_STOP) AND
ST02_Main.State = STATE_WAIT
END_TRANSITION

TRANSITION AutoRun:
ModeSelect.Mode=MODE_AUTO_RUN OR
ModeSelect.Mode=MODE_STEP_RUN
	OR (SpecialMode06.State=State_Run AND
		(gTypeCode=312 OR			(*93pol*)
		gTypeCode=499 OR				(*102pol*)
		gTypeCode=322))				(*160pol*)
END_TRANSITION

TRANSITION AutoStop:
(ModeSelect.Mode=MODE_AUTO_STOP OR
ModeSelect.Mode=MODE_STEP_STOP) AND
ST02_Main.State = STATE_WAIT
END_TRANSITION

TRANSITION #StateOK:
    Robot01.State=STATE_OK
AND gTipImp
END_TRANSITION
END_PROGRAM

(* POU zLibrary/ept/Funktionen/FB_CurrentStepHistorie, ST *)
FUNCTION_BLOCK FB_CurrentStepHistorie
VAR_INPUT
	st_CurrentStep	:STRING(20);
END_VAR

VAR
	arr_last_step_history 		:ARRAY[0..maxNumberOfPuffer] OF STRING;
	fb_Time					:TON;
	st_Time					:STRING;
	st_CurrentStepCopy		:STRING;
END_VAR
VAR_TEMP
	i					:INT;
END_VAR
VAR CONSTANT
	maxNumberOfPuffer			: INT:=30;
END_VAR
(*======================================================
   PRG: ST_CurrentStepHistorie
 ------------------------------------------------------
   Auth: 		Werner Friedl    						 
   Date: 		1.6.2015    						     
   Rev.: 		1.0	
   Desc:		Ablauf wird in einer Historie aufgezeichnet
   Historie:   1.0

	Beispiel eines Aufrufs:
	ST02_Nest05.FB_CurrentStepHistorie(st_CurrentStep:=ST02_Nest05.SFCCurrentStep);
 ========================================================*)

fb_Time();

IF st_CurrentStep<>st_CurrentStepCopy THEN
	fb_Time(IN:=FALSE);
	FOR i:=maxNumberOfPuffer TO 1  BY -1 DO
			arr_last_step_history[i] :=arr_last_step_history[i-1];
	END_FOR
	st_CurrentStepCopy:=st_CurrentStep;
	fb_Time(IN:=TRUE,PT:=t#100m);
END_IF
st_Time:=TIME_TO_STRING(fb_Time.ET);
st_Time:=DELETE(st_Time,2,1);
st_Time:=CONCAT(st_Time,': ');
arr_last_step_history[0]:=CONCAT(st_Time,st_CurrentStep);
END_FUNCTION_BLOCK

(* POU Stations/ST_00/ST00_SFCs/_SpecialModeSFCs/SpecialMode06, SFC *)
PROGRAM SpecialMode06 (*Used for: Dummytestprogramm*)
(* Date: 06.03.2019    Author: Rid Tobias   *)

VAR_OUTPUT
	SFCCurrentPOU		: STRING:='SpecialMode06';
	SFCCurrentStep		: STRING:='';
	SFCTime			: DINT;
 	State   				: DINT;
  	Result  				: DINT;
END_VAR
VAR_INPUT
	Start					: BOOL;

END_VAR
VAR

	MsgOK				: BOOL;
	MsgCancel			: BOOL;
	SFCRun				: BOOL;
	SFCTimeStart		: TIME;
  	LoopCounter   		: DINT;	(* aktuelle Dummynummer *)
	Delay				: TON;
	(*PartOk				: BOOL;	(* Ergebnisvariable für aktuelles *)*)
  	Dummy_ResOK		: BOOL;	(* Ergebnisvariable für den kompletten Dummytest *)
 	i           				: DINT;
  	NokMsgString		: STRING(255);
	startBand			:BOOL;
	NokMsgString1		 : STRING;

	StartErlaubt93pol			:BOOL;
	(* Userdefinded area *)

END_VAR
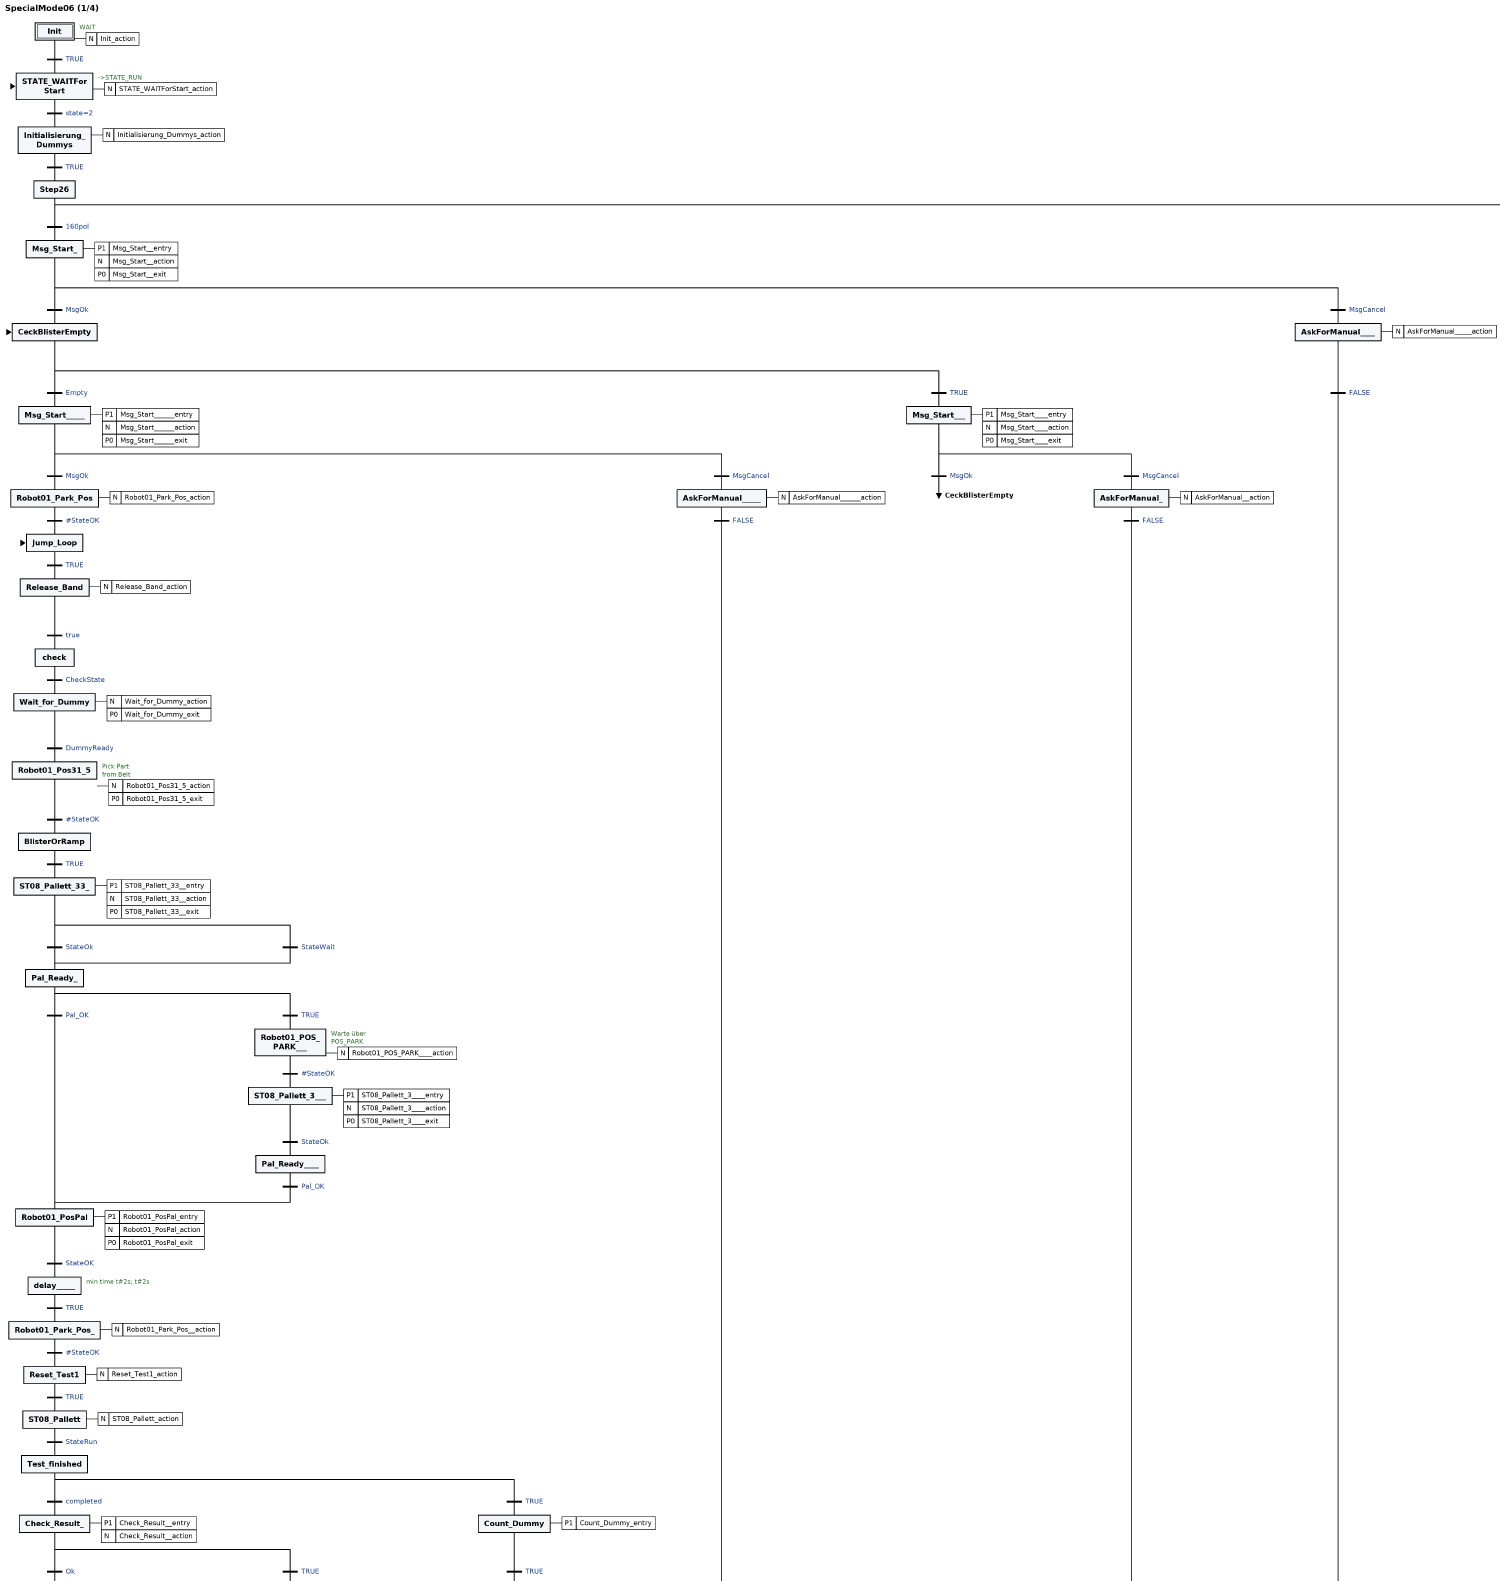
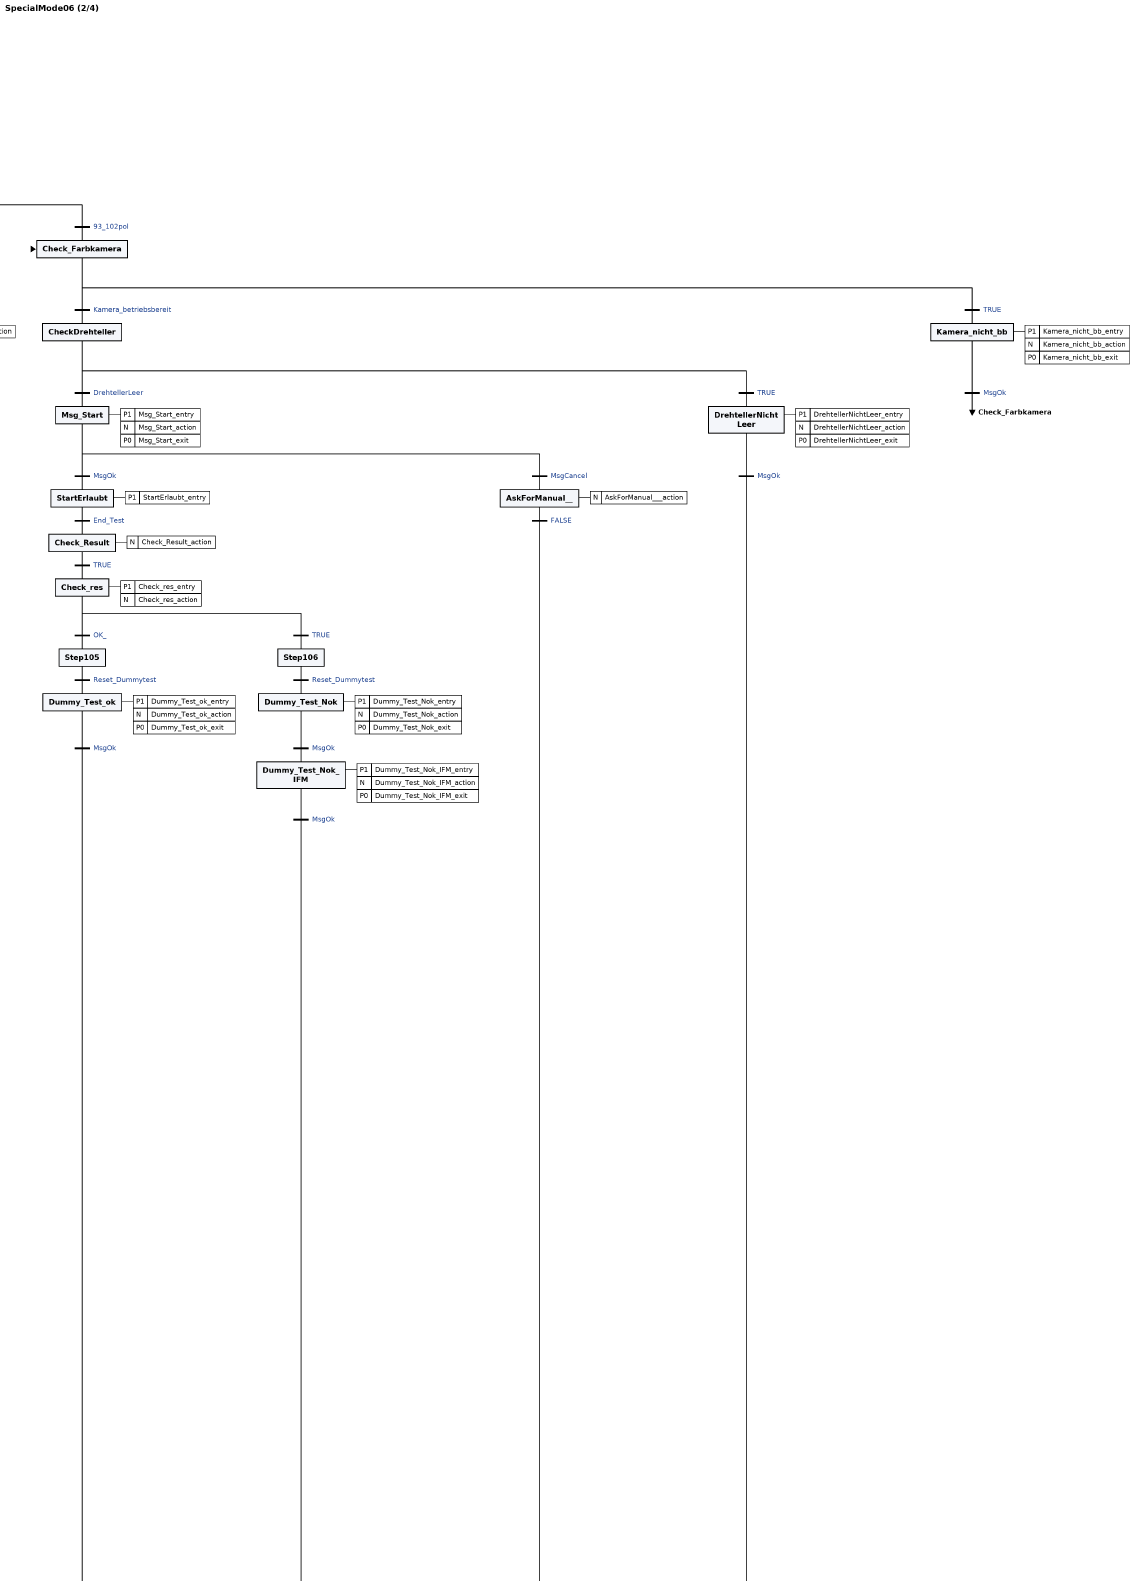
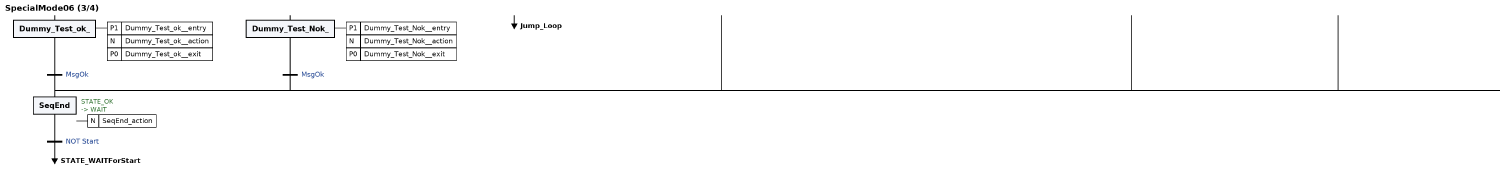
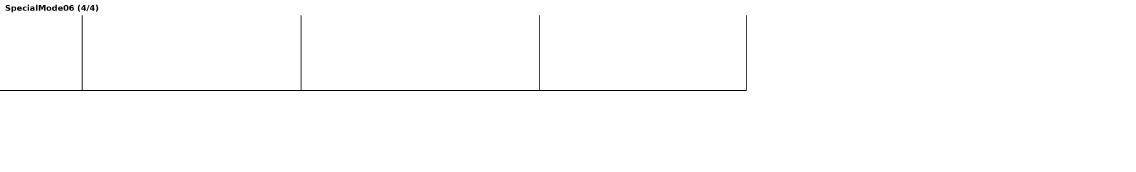
INITIAL_STEP Init: (* WAIT *)
	Init_action(N);
END_STEP
TRANSITION FROM Init TO STATE_WAITForStart := TRUE;
END_TRANSITION
STEP STATE_WAITForStart: (* ->STATE_RUN *)
	STATE_WAITForStart_action(N);
END_STEP
TRANSITION FROM STATE_WAITForStart TO Initialisierung_Dummys := state=2;
END_TRANSITION
STEP Initialisierung_Dummys:
	Initialisierung_Dummys_action(N);
END_STEP
TRANSITION FROM Initialisierung_Dummys TO Step26 := TRUE;
END_TRANSITION
STEP Step26:
END_STEP
TRANSITION FROM Step26 TO Msg_Start_ := 160pol;
END_TRANSITION
TRANSITION FROM Step26 TO Check_Farbkamera := 93_102pol;
END_TRANSITION
STEP Msg_Start_:
	Msg_Start__entry(P1);
	Msg_Start__action(N);
	Msg_Start__exit(P0);
END_STEP
TRANSITION FROM Msg_Start_ TO CeckBlisterEmpty := MsgOk;
END_TRANSITION
TRANSITION FROM Msg_Start_ TO AskForManual____ := MsgCancel;
END_TRANSITION
STEP CeckBlisterEmpty:
END_STEP
TRANSITION FROM CeckBlisterEmpty TO Msg_Start_____ := Empty;
END_TRANSITION
TRANSITION FROM CeckBlisterEmpty TO Msg_Start___ := TRUE;
END_TRANSITION
STEP Msg_Start___:
	Msg_Start____entry(P1);
	Msg_Start____action(N);
	Msg_Start____exit(P0);
END_STEP
TRANSITION FROM Msg_Start___ TO CeckBlisterEmpty := MsgOk;
END_TRANSITION
TRANSITION FROM Msg_Start___ TO AskForManual_ := MsgCancel;
END_TRANSITION
STEP AskForManual_:
	AskForManual__action(N);
END_STEP
TRANSITION FROM AskForManual_ TO SeqEnd := FALSE;
END_TRANSITION
STEP AskForManual____:
	AskForManual_____action(N);
END_STEP
TRANSITION FROM AskForManual____ TO SeqEnd := FALSE;
END_TRANSITION
STEP Msg_Start_____:
	Msg_Start______entry(P1);
	Msg_Start______action(N);
	Msg_Start______exit(P0);
END_STEP
TRANSITION FROM Msg_Start_____ TO Robot01_Park_Pos := MsgOk;
END_TRANSITION
TRANSITION FROM Msg_Start_____ TO AskForManual_____ := MsgCancel;
END_TRANSITION
STEP AskForManual_____:
	AskForManual______action(N);
END_STEP
TRANSITION FROM AskForManual_____ TO SeqEnd := FALSE;
END_TRANSITION
STEP Robot01_Park_Pos:
	Robot01_Park_Pos_action(N);
END_STEP
TRANSITION FROM Robot01_Park_Pos TO Jump_Loop := #StateOK;
END_TRANSITION
STEP Check_Farbkamera:
END_STEP
TRANSITION FROM Check_Farbkamera TO CheckDrehteller := Kamera_betriebsbereit;
END_TRANSITION
TRANSITION FROM Check_Farbkamera TO Kamera_nicht_bb := TRUE;
END_TRANSITION
STEP CheckDrehteller:
END_STEP
TRANSITION FROM CheckDrehteller TO Msg_Start := DrehtellerLeer;
END_TRANSITION
TRANSITION FROM CheckDrehteller TO DrehtellerNichtLeer := TRUE;
END_TRANSITION
STEP DrehtellerNichtLeer:
	DrehtellerNichtLeer_entry(P1);
	DrehtellerNichtLeer_action(N);
	DrehtellerNichtLeer_exit(P0);
END_STEP
TRANSITION FROM DrehtellerNichtLeer TO SeqEnd := MsgOk;
END_TRANSITION
STEP Kamera_nicht_bb:
	Kamera_nicht_bb_entry(P1);
	Kamera_nicht_bb_action(N);
	Kamera_nicht_bb_exit(P0);
END_STEP
TRANSITION FROM Kamera_nicht_bb TO Check_Farbkamera := MsgOk;
END_TRANSITION
STEP Msg_Start:
	Msg_Start_entry(P1);
	Msg_Start_action(N);
	Msg_Start_exit(P0);
END_STEP
TRANSITION FROM Msg_Start TO StartErlaubt := MsgOk;
END_TRANSITION
TRANSITION FROM Msg_Start TO AskForManual__ := MsgCancel;
END_TRANSITION
STEP AskForManual__:
	AskForManual___action(N);
END_STEP
TRANSITION FROM AskForManual__ TO SeqEnd := FALSE;
END_TRANSITION
STEP StartErlaubt:
	StartErlaubt_entry(P1);
END_STEP
TRANSITION FROM StartErlaubt TO Check_Result := End_Test;
END_TRANSITION
STEP Check_Result:
	Check_Result_action(N);
END_STEP
TRANSITION FROM Check_Result TO Check_res := TRUE;
END_TRANSITION
STEP Check_res:
	Check_res_entry(P1);
	Check_res_action(N);
END_STEP
TRANSITION FROM Check_res TO Step105 := OK_;
END_TRANSITION
TRANSITION FROM Check_res TO Step106 := TRUE;
END_TRANSITION
STEP Step105:
END_STEP
TRANSITION FROM Step105 TO Dummy_Test_ok := Reset_Dummytest;
END_TRANSITION
STEP Dummy_Test_ok:
	Dummy_Test_ok_entry(P1);
	Dummy_Test_ok_action(N);
	Dummy_Test_ok_exit(P0);
END_STEP
TRANSITION FROM Dummy_Test_ok TO SeqEnd := MsgOk;
END_TRANSITION
STEP Step106:
END_STEP
TRANSITION FROM Step106 TO Dummy_Test_Nok := Reset_Dummytest;
END_TRANSITION
STEP Dummy_Test_Nok:
	Dummy_Test_Nok_entry(P1);
	Dummy_Test_Nok_action(N);
	Dummy_Test_Nok_exit(P0);
END_STEP
TRANSITION FROM Dummy_Test_Nok TO Dummy_Test_Nok_IFM := MsgOk;
END_TRANSITION
STEP Dummy_Test_Nok_IFM:
	Dummy_Test_Nok_IFM_entry(P1);
	Dummy_Test_Nok_IFM_action(N);
	Dummy_Test_Nok_IFM_exit(P0);
END_STEP
TRANSITION FROM Dummy_Test_Nok_IFM TO SeqEnd := MsgOk;
END_TRANSITION
STEP Jump_Loop:
END_STEP
TRANSITION FROM Jump_Loop TO Release_Band := TRUE;
END_TRANSITION
STEP Release_Band:
	Release_Band_action(N);
END_STEP
TRANSITION FROM Release_Band TO check := true;
END_TRANSITION
STEP check:
END_STEP
TRANSITION FROM check TO Wait_for_Dummy := CheckState;
END_TRANSITION
STEP Wait_for_Dummy:
	Wait_for_Dummy_action(N);
	Wait_for_Dummy_exit(P0);
END_STEP
TRANSITION FROM Wait_for_Dummy TO Robot01_Pos31_5 := DummyReady;
END_TRANSITION
STEP Robot01_Pos31_5: (* Pick Part / from Belt *)
	Robot01_Pos31_5_action(N);
	Robot01_Pos31_5_exit(P0);
END_STEP
TRANSITION FROM Robot01_Pos31_5 TO BlisterOrRamp := #StateOK;
END_TRANSITION
STEP BlisterOrRamp:
END_STEP
TRANSITION FROM BlisterOrRamp TO ST08_Pallett_33_ := TRUE;
END_TRANSITION
STEP ST08_Pallett_33_:
	ST08_Pallett_33__entry(P1);
	ST08_Pallett_33__action(N);
	ST08_Pallett_33__exit(P0);
END_STEP
TRANSITION FROM ST08_Pallett_33_ TO Pal_Ready_ := StateOk;
END_TRANSITION
TRANSITION FROM ST08_Pallett_33_ TO Pal_Ready_ := StateWait;
END_TRANSITION
STEP Pal_Ready_:
END_STEP
TRANSITION FROM Pal_Ready_ TO Robot01_PosPal := Pal_OK;
END_TRANSITION
TRANSITION FROM Pal_Ready_ TO Robot01_POS_PARK___ := TRUE;
END_TRANSITION
STEP Robot01_POS_PARK___: (* Warte über / POS_PARK *)
	Robot01_POS_PARK____action(N);
END_STEP
TRANSITION FROM Robot01_POS_PARK___ TO ST08_Pallett_3___ := #StateOK;
END_TRANSITION
STEP ST08_Pallett_3___:
	ST08_Pallett_3____entry(P1);
	ST08_Pallett_3____action(N);
	ST08_Pallett_3____exit(P0);
END_STEP
TRANSITION FROM ST08_Pallett_3___ TO Pal_Ready____ := StateOk;
END_TRANSITION
STEP Pal_Ready____:
END_STEP
TRANSITION FROM Pal_Ready____ TO Robot01_PosPal := Pal_OK;
END_TRANSITION
STEP Robot01_PosPal:
	Robot01_PosPal_entry(P1);
	Robot01_PosPal_action(N);
	Robot01_PosPal_exit(P0);
END_STEP
TRANSITION FROM Robot01_PosPal TO delay_____ := StateOK;
END_TRANSITION
STEP delay_____: (* min time t#2s; t#2s *)
END_STEP
TRANSITION FROM delay_____ TO Robot01_Park_Pos_ := TRUE;
END_TRANSITION
STEP Robot01_Park_Pos_:
	Robot01_Park_Pos__action(N);
END_STEP
TRANSITION FROM Robot01_Park_Pos_ TO Reset_Test1 := #StateOK;
END_TRANSITION
STEP Reset_Test1:
	Reset_Test1_action(N);
END_STEP
TRANSITION FROM Reset_Test1 TO ST08_Pallett := TRUE;
END_TRANSITION
STEP ST08_Pallett:
	ST08_Pallett_action(N);
END_STEP
TRANSITION FROM ST08_Pallett TO Test_finished := StateRun;
END_TRANSITION
STEP Test_finished:
END_STEP
TRANSITION FROM Test_finished TO Check_Result_ := completed;
END_TRANSITION
TRANSITION FROM Test_finished TO Count_Dummy := TRUE;
END_TRANSITION
STEP Count_Dummy:
	Count_Dummy_entry(P1);
END_STEP
TRANSITION FROM Count_Dummy TO Jump_Loop := TRUE;
END_TRANSITION
STEP Check_Result_:
	Check_Result__entry(P1);
	Check_Result__action(N);
END_STEP
TRANSITION FROM Check_Result_ TO Dummy_Test_ok_ := Ok;
END_TRANSITION
TRANSITION FROM Check_Result_ TO Dummy_Test_Nok_ := TRUE;
END_TRANSITION
STEP Dummy_Test_Nok_:
	Dummy_Test_Nok__entry(P1);
	Dummy_Test_Nok__action(N);
	Dummy_Test_Nok__exit(P0);
END_STEP
TRANSITION FROM Dummy_Test_Nok_ TO SeqEnd := MsgOk;
END_TRANSITION
STEP Dummy_Test_ok_:
	Dummy_Test_ok__entry(P1);
	Dummy_Test_ok__action(N);
	Dummy_Test_ok__exit(P0);
END_STEP
TRANSITION FROM Dummy_Test_ok_ TO SeqEnd := MsgOk;
END_TRANSITION
STEP SeqEnd: (* STATE_OK / -> WAIT *)
	SeqEnd_action(N);
END_STEP
TRANSITION FROM SeqEnd TO STATE_WAITForStart := NOT Start;
END_TRANSITION

ACTION Init_action:
Start:=FALSE;
State:=STATE_WAIT;
LoopCounter:=1;
startBand := FALSE;
StartErlaubt93pol:=FALSE;
END_ACTION

ACTION STATE_WAITForStart_action:
IF Start=TRUE
THEN
	State:=STATE_RUN;
	Result:=RESULT_NON;
	SFCTimeStart:=TIME();
(*ELSE*)
END_IF
END_ACTION

ACTION Initialisierung_Dummys_action:
(*Reihenfolge der Dummys für 160 pol.*)
(*		TRUE = Gutteil
   		FALSE = Schlechtteil		*)
Dummy_test_Vorgabe[1] := FALSE;
Dummy_test_Vorgabe[2] := FALSE;
Dummy_test_Vorgabe[3] := FALSE;
Dummy_test_Vorgabe[4] := FALSE;
Dummy_test_Vorgabe[5] := FALSE;
Dummy_test_Vorgabe[6] := FALSE;
END_ACTION

ACTION Msg_Start__entry:
MessageHandler.ClearMessageLines(sVisu:=Visu.Message);
END_ACTION

ACTION Msg_Start__action:
MessageHandler.Msg.ID:='PM59';
MessageHandler.Msg.Name:='Prüfung Dummy/Nio-Teile';
MessageHandler.Msg.Text:='Blister und Band leer räumen und$R$N Teile im Blister auf 0 stellen$R$NJa: Start mit OK$R$NNein: Abbrechen';
MessageHandler.Msg.Color:=Color.yellow;
MessageHandler.Msg.Station:=0;


MessageHandler(
	Prio:=2, 									(*1=highest, .. , 4=lowest*)
	Btn1Addr:=ADR(MsgOk),			(*Address of Button1 , if Zero then Button is unvisible*)
	Btn2Addr:=ADR(MsgCancel),	(*Address of Button2 , if Zero then Button is unvisible*)
	sVisu:=Visu.Message);
END_ACTION

ACTION Msg_Start__exit:
MsgOk:=FALSE;
MsgCancel:=FALSE;
END_ACTION

ACTION Msg_Start____entry:
MessageHandler.ClearMessageLines(sVisu:=Visu.Message);
END_ACTION

ACTION Msg_Start____action:
MessageHandler.Msg.ID:='PM60';
MessageHandler.Msg.Name:='Prüfung Dummy/Nio-Teile';
MessageHandler.Msg.Text:='Blister ist nicht leer, Blister leerräumen 0$R$N und Teile auf Anzahl Teile auf 0 stellen$R$NJa: Start mit OK$R$NNein: Abbrechen';
MessageHandler.Msg.Color:=Color.yellow;
MessageHandler.Msg.Station:=0;


MessageHandler(
	Prio:=2, 									(*1=highest, .. , 4=lowest*)
	Btn1Addr:=ADR(MsgOk),			(*Address of Button1 , if Zero then Button is unvisible*)
	Btn2Addr:=ADR(MsgCancel),	(*Address of Button2 , if Zero then Button is unvisible*)
	sVisu:=Visu.Message);
END_ACTION

ACTION Msg_Start____exit:
MsgOk:=FALSE;
MsgCancel:=FALSE;
END_ACTION

ACTION AskForManual__action:
ModeSelect.AskForManual:=TRUE;
END_ACTION

ACTION AskForManual_____action:
ModeSelect.AskForManual:=TRUE;
END_ACTION

ACTION Msg_Start______entry:
MessageHandler.ClearMessageLines(sVisu:=Visu.Message);
END_ACTION

ACTION Msg_Start______action:
MessageHandler.Msg.ID:='PM57';
MessageHandler.Msg.Name:='Prüfung Dummy/Nio-Teile';
MessageHandler.Msg.Text:='Bitte die 6 Prüfteile nacheinander einlegen$R$NJedes Teil muss mit Ok bestätigt werden$R$NJa: Start mit OK$R$NNein: Abbrechen';
MessageHandler.Msg.Color:=Color.yellow;
MessageHandler.Msg.Station:=0;


MessageHandler(
	Prio:=2, 									(*1=highest, .. , 4=lowest*)
	Btn1Addr:=ADR(MsgOk),			(*Address of Button1 , if Zero then Button is unvisible*)
	Btn2Addr:=ADR(MsgCancel),	(*Address of Button2 , if Zero then Button is unvisible*)
	sVisu:=Visu.Message);
END_ACTION

ACTION Msg_Start______exit:
MsgOk:=FALSE;
MsgCancel:=FALSE;
END_ACTION

ACTION AskForManual______action:
ModeSelect.AskForManual:=TRUE;
END_ACTION

ACTION Robot01_Park_Pos_action:
Robot01.PosNo:=POS_PARK;
Robot01.PosOffset:=gRobotOffset;
Robot01.Override:=MP.ST00.Override;
Robot01.SetToolOn:=TRUE;
Robot01.SetToolOff:=FALSE;
Robot01.ExecuteMove:=TRUE;
END_ACTION

ACTION DrehtellerNichtLeer_entry:
MessageHandler.ClearMessageLines(sVisu:=Visu.Message);
END_ACTION

ACTION DrehtellerNichtLeer_action:
MessageHandler.Msg.ID:='PM63';
MessageHandler.Msg.Name:='Check Drehteller';
MessageHandler.Msg.Text:='Drehteller ist nicht Leer';
MessageHandler.Msg.Color:=Color.red;
MessageHandler.Msg.Station:=1;


MessageHandler(
	Prio:=2, 							(*1=highest, .. , 4=lowest*)
	Btn1Addr:=ADR(MsgOk),			(*Address of Button1 , if Zero then Button is unvisible*)
	Btn2Addr:=,						(*Address of Button2 , if Zero then Button is unvisible*)
	sVisu:=Visu.Message);
END_ACTION

ACTION DrehtellerNichtLeer_exit:
MsgOk:=FALSE;
MsgCancel:=FALSE;
ST02_DT_95_A1.b_quitt:=TRUE;
END_ACTION

ACTION Kamera_nicht_bb_entry:
MessageHandler.ClearMessageLines(sVisu:=Visu.Message);
END_ACTION

ACTION Kamera_nicht_bb_action:
MessageHandler.Msg.ID:='PM62';
MessageHandler.Msg.Name:='Check Camera';
MessageHandler.Msg.Text:='Sesopart Kamera ist nicht betriebsbereit';
MessageHandler.Msg.Color:=Color.red;
MessageHandler.Msg.Station:=1;


MessageHandler(
	Prio:=2, 							(*1=highest, .. , 4=lowest*)
	Btn1Addr:=ADR(MsgOk),			(*Address of Button1 , if Zero then Button is unvisible*)
	Btn2Addr:=,						(*Address of Button2 , if Zero then Button is unvisible*)
	sVisu:=Visu.Message);
END_ACTION

ACTION Kamera_nicht_bb_exit:
MsgOk:=FALSE;
MsgCancel:=FALSE;
ST02_DT_95_A1.b_quitt:=TRUE;
END_ACTION

ACTION Msg_Start_entry:
MessageHandler.ClearMessageLines(sVisu:=Visu.Message);
END_ACTION

ACTION Msg_Start_action:
MessageHandler.Msg.ID:='PM58';
MessageHandler.Msg.Name:='Prüfung Dummy/Nio-Teile';
MessageHandler.Msg.Text:='Bitte Drehteller leer machen dann $R$Ndie 6 Prüfteile nacheinander einlegen$R$NJa: Start mit OK$R$NNein: Abbrechen';
MessageHandler.Msg.Color:=Color.yellow;
MessageHandler.Msg.Station:=0;


MessageHandler(
	Prio:=2, 									(*1=highest, .. , 4=lowest*)
	Btn1Addr:=ADR(MsgOk),			(*Address of Button1 , if Zero then Button is unvisible*)
	Btn2Addr:=ADR(MsgCancel),	(*Address of Button2 , if Zero then Button is unvisible*)
	sVisu:=Visu.Message);
END_ACTION

ACTION Msg_Start_exit:
MsgOk:=FALSE;
MsgCancel:=FALSE;
END_ACTION

ACTION AskForManual___action:
ModeSelect.AskForManual:=TRUE;
END_ACTION

ACTION StartErlaubt_entry:
StartErlaubt93pol:=TRUE;
END_ACTION

ACTION Check_Result_action:
(*Erklärung der Auswertung:
In der Produktion wird  nur OK und NOK ausgwertet:
   0 = Teil noch nicht bearbeitet bzw. Nest leer
   1 =  Druck ist OK
   9 = Druck ist NOK
Bei der Dummyprüfung muss passend zum Dummy rot, blau oder beide NOK sein:
   6= Teil roter und blauer Druck NOK ist nur bei der Dummyprüfung aktiv
   7= Teil roter Druck NOKist nur bei der Dummyprüfung aktiv
   8= Teil blauer Druck NOK ist nur bei der Dummyprüfung aktiv
Lage:	
Ziffer 1 = 90°		Ziffer 2 =180°
*)

(*Dummy1*)
IF ST02_Main.ResultBuffer[6] = 78 THEN
	 Mp.ST02.Dummy_test_Result[1] := TRUE;
ELSE
	 Mp.ST02.Dummy_test_Result[1] := FALSE;
END_IF
(*Dummy2*)
IF ST02_Main.ResultBuffer[5] = 11 THEN
	 Mp.ST02.Dummy_test_Result[2] :=  TRUE;
ELSE
	 Mp.ST02.Dummy_test_Result[2] := FALSE;
END_IF
(*Dummy3*)
IF ST02_Main.ResultBuffer[4] = 16 THEN
	 Mp.ST02.Dummy_test_Result[3] :=  TRUE;
ELSE
	 Mp.ST02.Dummy_test_Result[3] := FALSE;
END_IF
(*Dummy4*)
IF ST02_Main.ResultBuffer[3] = 66 THEN
	 Mp.ST02.Dummy_test_Result[4] :=  TRUE;
ELSE
	 Mp.ST02.Dummy_test_Result[4] := FALSE;
END_IF
(*Dummy5*)
IF ST02_Main.ResultBuffer[2] = 66 THEN
	 Mp.ST02.Dummy_test_Result[5] :=  TRUE;
ELSE
	 Mp.ST02.Dummy_test_Result[5] := FALSE;
END_IF
(*Dummy6*)
IF ST02_Main.ResultBuffer[1] = 11 THEN
	 Mp.ST02.Dummy_test_Result[6] := TRUE;
ELSE
	 Mp.ST02.Dummy_test_Result[6] := FALSE;
END_IF


(*IFM Flügelerkennung*)
IF ST03_102pol_Zufuehrung.ResultBufferIFM[6] = TRUE THEN
	  Mp.ST02.Dummy_test_Result[7]  := TRUE;
ELSE
	 Mp.ST02.Dummy_test_Result[7] := FALSE;
END_IF

IF ST03_102pol_Zufuehrung.ResultBufferIFM[5] = TRUE THEN
	 Mp.ST02.Dummy_test_Result[8] :=  TRUE;
ELSE
	 Mp.ST02.Dummy_test_Result[8] := FALSE;
END_IF


IF ST03_102pol_Zufuehrung.ResultBufferIFM[4] = FALSE THEN
	 Mp.ST02.Dummy_test_Result[9] :=  TRUE;
ELSE
	 Mp.ST02.Dummy_test_Result[9] := FALSE;
END_IF


IF ST03_102pol_Zufuehrung.ResultBufferIFM[3] = FALSE THEN
	 Mp.ST02.Dummy_test_Result[10] :=  TRUE;
ELSE
	 Mp.ST02.Dummy_test_Result[10] := FALSE;
END_IF


IF ST03_102pol_Zufuehrung.ResultBufferIFM[2] = TRUE THEN
	 Mp.ST02.Dummy_test_Result[11] :=  TRUE;
ELSE
	 Mp.ST02.Dummy_test_Result[11] := FALSE;
END_IF


IF ST03_102pol_Zufuehrung.ResultBufferIFM[1] = FALSE THEN
	 Mp.ST02.Dummy_test_Result[12] := TRUE;
ELSE
	 Mp.ST02.Dummy_test_Result[12] := FALSE;
END_IF
END_ACTION

ACTION Check_res_entry:
Dummy_ResOK:=TRUE;
END_ACTION

ACTION Check_res_action:
FOR i:=1 TO 12
	DO
	  IF Mp.ST02.Dummy_test_Result[i] = FALSE
	  THEN
	     Dummy_ResOK:=FALSE;
	  END_IF
END_FOR
END_ACTION

ACTION Dummy_Test_ok_entry:
MessageHandler.ClearMessageLines(sVisu:=Visu.Message);
MsgOk:=FALSE;
END_ACTION

ACTION Dummy_Test_ok_action:
MessageHandler.Msg.ID:='PM54';
MessageHandler.Msg.Name:='DummyTest';
MessageHandler.Msg.Text:=' Dummy Pruefung OK, Ergebnis aller Teile OK ';
MessageHandler.Msg.Color:=Color.green;
MessageHandler.Msg.Station:=1;


MessageHandler(
	Prio:=2, 								(*1=highest, .. , 4=lowest*)
	Btn1Addr:=ADR(MsgOk),						(*Address of Button1 , if Zero then Button is unvisible*)
	Btn2Addr:=0,						(*Address of Button2 , if Zero then Button is unvisible*)
	sVisu:=Visu.Message);
END_ACTION

ACTION Dummy_Test_ok_exit:
MessageHandler.ClearMessageLines(sVisu:=Visu.Message);
MsgOk:=FALSE;
END_ACTION

ACTION Dummy_Test_Nok_entry:
MessageHandler.ClearMessageLines(sVisu:=Visu.Message);
MsgOk:=FALSE;
END_ACTION

ACTION Dummy_Test_Nok_action:
NokMsgString:='';
NokMsgString1:='';

MessageHandler.Msg.ID:='PM55';
MessageHandler.Msg.Name:='Sensopart Dummyprüfung NOK';
MessageHandler.Msg.Text:=CONCAT(NokMsgString,'$N$R');
MessageHandler.Msg.Text:=CONCAT(MessageHandler.Msg.Text,NokMsgString1);
MessageHandler.Msg.Color:=Color.red;
MessageHandler.Msg.Station:=2;

FOR i:= 1 TO 6 BY 1 DO
	MessageHandler.MessageLine[i].MsgTypeEnum:=MsgDataTypeString;
	MessageHandler.MessageLine[i].Text:=CONCAT('Dummy_',DINT_TO_STRING(i));
	IF Mp.ST02.Dummy_test_Result[i] THEN
		MessageHandler.MessageLine[i].MsgString:='OK';
	ELSE
		MessageHandler.MessageLine[i].MsgString:='NOK';
	END_IF
END_FOR

MessageHandler(
	Prio:=2, 								(*1=highest, .. , 4=lowest*)
	Btn1Addr:=ADR(MsgOk),						(*Address of Button1 , if Zero then Button is unvisible*)
	Btn2Addr:=0,						(*Address of Button2 , if Zero then Button is unvisible*)
	sVisu:=Visu.Message);
END_ACTION

ACTION Dummy_Test_Nok_exit:
MessageHandler.ClearMessageLines(sVisu:=Visu.Message);
MsgOk:=FALSE;
END_ACTION

ACTION Dummy_Test_Nok_IFM_entry:
MessageHandler.ClearMessageLines(sVisu:=Visu.Message);
MsgOk:=FALSE;
END_ACTION

ACTION Dummy_Test_Nok_IFM_action:
NokMsgString:='';
NokMsgString1:='';

MessageHandler.Msg.ID:='PM56';
MessageHandler.Msg.Name:='IFM Dummyprüfung NOK';
MessageHandler.Msg.Text:='IFM Dummyprüfung NOK';
MessageHandler.Msg.Color:=Color.red;
MessageHandler.Msg.Station:=2;


FOR i:= 7 TO 12 BY 1 DO
	MessageHandler.MessageLine[i-6].MsgTypeEnum:=MsgDataTypeString;
	MessageHandler.MessageLine[i-6].Text:=CONCAT('Dummy_',DINT_TO_STRING(i));
	IF Mp.ST02.Dummy_test_Result[i] THEN
		MessageHandler.MessageLine[i-6].MsgString:='OK';
	ELSE
		MessageHandler.MessageLine[i-6].MsgString:='NOK';
	END_IF
END_FOR


MessageHandler(
	Prio:=2, 								(*1=highest, .. , 4=lowest*)
	Btn1Addr:=ADR(MsgOk),						(*Address of Button1 , if Zero then Button is unvisible*)
	Btn2Addr:=0,						(*Address of Button2 , if Zero then Button is unvisible*)
	sVisu:=Visu.Message);
END_ACTION

ACTION Dummy_Test_Nok_IFM_exit:
MessageHandler.ClearMessageLines(sVisu:=Visu.Message);
MsgOk:=FALSE;
END_ACTION

ACTION Release_Band_action:
ST03_160pol_Zufuehrung.Start:=TRUE;
startBand := TRUE;
END_ACTION

ACTION Wait_for_Dummy_action:
Delay.IN:=ST03_422_B64_4.BitInToCheck;  		 (* Schnittstelle Bedrucken Tinte ISK i.O. oder n.i.O. auf Übergabeposition *)
END_ACTION

ACTION Wait_for_Dummy_exit:
(*Auswertung Kamera Ergebnis für die 6 Dummys*)
IF NOT MP.ST03.SGM_3621 THEN
	IF LoopCounter = 1 THEN
		IF 	ST03_160pol_Zufuehrung.CamResult = 11 AND
			ST03_160pol_Zufuehrung.CamResult2 = 11	 AND
			ST03_160pol_Zufuehrung.CamResult3 = 11 THEN
			Dummy_test_Result[1] := TRUE;
		ELSE
			Dummy_test_Result[1] := FALSE;
		END_IF
	ELSIF LoopCounter = 2 THEN
		IF 	ST03_160pol_Zufuehrung.CamResult = 11 AND
			ST03_160pol_Zufuehrung.CamResult2 = 11  AND
			ST03_160pol_Zufuehrung.CamResult3 = 11 THEN
			Dummy_test_Result[2] := TRUE;
		ELSE
			Dummy_test_Result[2] := FALSE;
		END_IF
	ELSIF LoopCounter = 3 THEN
		IF 	ST03_160pol_Zufuehrung.CamResult = 99 AND
			ST03_160pol_Zufuehrung.CamResult2 = 99	 AND
			ST03_160pol_Zufuehrung.CamResult3 = 99 THEN
			Dummy_test_Result[3] := TRUE;
		ELSE
			Dummy_test_Result[3] := FALSE;
		END_IF
	
	ELSIF LoopCounter = 4 THEN
		IF 	ST03_160pol_Zufuehrung.CamResult = 11 AND
			ST03_160pol_Zufuehrung.CamResult2 = 11	 AND
			ST03_160pol_Zufuehrung.CamResult3 = 99 THEN
			Dummy_test_Result[4] := TRUE;
		ELSE
			Dummy_test_Result[4] := FALSE;
		END_IF
	
	
	ELSIF LoopCounter = 5 THEN
		IF 	ST03_160pol_Zufuehrung.CamResult = 99 AND
			ST03_160pol_Zufuehrung.CamResult2 = 99	 AND
			ST03_160pol_Zufuehrung.CamResult3 = 99 THEN
			Dummy_test_Result[5] := TRUE;
		ELSE
			Dummy_test_Result[5] := FALSE;
		END_IF
	
	ELSIF LoopCounter = 6 THEN
		IF 	ST03_160pol_Zufuehrung.CamResult = 99 AND
			ST03_160pol_Zufuehrung.CamResult2 = 99	 AND
			ST03_160pol_Zufuehrung.CamResult3 = 99 THEN
			Dummy_test_Result[6] := TRUE;
		ELSE
			Dummy_test_Result[6] := FALSE;
		END_IF
	END_IF
ELSE
	IF LoopCounter = 1 THEN
		IF 	ST03_160pol_Zufuehrung.CamResult = 11 AND
			ST03_160pol_Zufuehrung.CamResult2 = 11	 AND
			ST03_160pol_Zufuehrung.CamResult3 = 11 THEN
			Dummy_test_Result[1] := TRUE;
		ELSE
			Dummy_test_Result[1] := FALSE;
		END_IF
	ELSIF LoopCounter = 2 THEN
		IF 	ST03_160pol_Zufuehrung.CamResult = 11 AND
			ST03_160pol_Zufuehrung.CamResult2 = 11	 AND
			ST03_160pol_Zufuehrung.CamResult3 = 11 THEN
			Dummy_test_Result[2] := TRUE;
		ELSE
			Dummy_test_Result[2] := FALSE;
		END_IF
	ELSIF LoopCounter = 3 THEN
		IF 	ST03_160pol_Zufuehrung.CamResult = 99 AND
			ST03_160pol_Zufuehrung.CamResult2 = 99	 AND
			ST03_160pol_Zufuehrung.CamResult3 = 99 THEN
			Dummy_test_Result[3] := TRUE;
		ELSE
			Dummy_test_Result[3] := FALSE;
		END_IF
	
	ELSIF LoopCounter = 4 THEN
		IF 	ST03_160pol_Zufuehrung.CamResult = 11 AND
			ST03_160pol_Zufuehrung.CamResult2 = 11	 AND
			ST03_160pol_Zufuehrung.CamResult3 = 99 THEN
			Dummy_test_Result[4] := TRUE;
		ELSE
			Dummy_test_Result[4] := FALSE;
		END_IF
	
	
	ELSIF LoopCounter = 5 THEN
		IF 	ST03_160pol_Zufuehrung.CamResult =  99 AND
			ST03_160pol_Zufuehrung.CamResult2 = 99	 AND
			ST03_160pol_Zufuehrung.CamResult3 = 99 THEN
			Dummy_test_Result[5] := TRUE;
		ELSE
			Dummy_test_Result[5] := FALSE;
		END_IF
	
	ELSIF LoopCounter = 6 THEN
		IF	ST03_160pol_Zufuehrung.CamResult = 99 AND
			ST03_160pol_Zufuehrung.CamResult2 = 99 AND
			ST03_160pol_Zufuehrung.CamResult3 = 99 THEN
			Dummy_test_Result[6] := TRUE;
		ELSE
			Dummy_test_Result[6] := FALSE;
		END_IF
	END_IF
END_IF
END_ACTION

ACTION Robot01_Pos31_5_action:
Robot01.PosNo:=POS_WT_POS1;
Robot01.PosOffset:=gRobotOffset;
Robot01.Override:=MP.ST00.Override;
Robot01.SetToolOn:=FALSE;
Robot01.SetToolOff:=TRUE;
Robot01.ExecuteMove:=TRUE;
END_ACTION

ACTION Robot01_Pos31_5_exit:
IF ST03_160pol_Zufuehrung.PartOk THEN
	gRob01GripState:=PART_OK;
ELSE
	gRob01GripState:=PART_NOK;
END_IF
END_ACTION

ACTION ST08_Pallett_33__entry:
ProcessMessage01:='';
END_ACTION

ACTION ST08_Pallett_33__action:
ProcessMessage01:='1IM7';(*warte Pallette*)
END_ACTION

ACTION ST08_Pallett_33__exit:
ST08_Process.Start:=FALSE;
ProcessMessage01:='';
END_ACTION

ACTION Robot01_POS_PARK____action:
Robot01.PosNo:=POS_PARK;
Robot01.PosOffset:=gRobotOffset;
Robot01.Override:=MP.ST00.Override;
Robot01.SetToolOn:=FALSE;
Robot01.SetToolOff:=FALSE;
Robot01.ExecuteMove:=TRUE;
END_ACTION

ACTION ST08_Pallett_3____entry:
ProcessMessage01:='';
END_ACTION

ACTION ST08_Pallett_3____action:
ProcessMessage01:='1IM7';(*warte Pallette*)
END_ACTION

ACTION ST08_Pallett_3____exit:
ST08_Process.Start:=FALSE;
ProcessMessage01:='';
END_ACTION

ACTION Robot01_PosPal_entry:
IF 	PosIdx<TD.PartsInRoboGripper THEN
	PosIdx:=TD.PartsInRoboGripper;
END_IF
END_ACTION

ACTION Robot01_PosPal_action:
Robot01.PosNo:=POS_FEED_PAL_WAIT + (PosIdx/TD.PartsInRoboGripper);
Robot01.PosOffset:=gRobotOffset;
Robot01.Override:=MP.ST00.Override;
Robot01.SetToolOn:=TRUE;
Robot01.SetToolOff:=FALSE;
Robot01.ExecuteMove:=TRUE;
END_ACTION

ACTION Robot01_PosPal_exit:
gRob01GripState:=PART_NO;
PosIdx:=PosIdx+TD.PartsInRoboGripper;
gPartsInserted:=gPartsInserted+TD.PartsInRoboGripper;
gPartsTest:=gPartsTest+TD.PartsInRoboGripper;
END_ACTION

ACTION Robot01_Park_Pos__action:
Robot01.PosNo:=POS_PARK;
Robot01.PosOffset:=gRobotOffset;
Robot01.Override:=MP.ST00.Override;
Robot01.SetToolOn:=FALSE;
Robot01.SetToolOff:=FALSE;
Robot01.ExecuteMove:=TRUE;
END_ACTION

ACTION Reset_Test1_action:
(*für das ausschleusen der Testteile mit einem Blister*)
IF LoopCounter >= MAX_NO_OF_DUMMYS THEN
	ST08_Palletizing.TestpartMoveOut:=TRUE;
END_IF
END_ACTION

ACTION ST08_Pallett_action:
IF 	ST08_Process.State=STATE_WAIT THEN
	ST08_Process.Start:=TRUE;
END_IF
END_ACTION

ACTION Count_Dummy_entry:
LoopCounter := LoopCounter +1;
END_ACTION

ACTION Check_Result__entry:
Dummy_ResOK:=TRUE;
END_ACTION

ACTION Check_Result__action:
(*Überprüfung, ob alle Dummys in der richtigen Reihenfolge waren*)
FOR i:=1 TO MAX_NO_OF_DUMMYS
DO
	IF Dummy_test_Result[i] = FALSE
	THEN
		Dummy_ResOK:=FALSE;
	END_IF
END_FOR
END_ACTION

ACTION Dummy_Test_Nok__entry:
MessageHandler.ClearMessageLines(sVisu:=Visu.Message);

NokMsgString:='';
END_ACTION

ACTION Dummy_Test_Nok__action:
MessageHandler.Msg.ID:='PM55';
MessageHandler.Msg.Name:='Dummyprüfung NOK';
MessageHandler.Msg.Text:='Dummyprüfung NOK';
MessageHandler.Msg.Color:=Color.red;
MessageHandler.Msg.Station:=2;


FOR i:= 1 TO MAX_NO_OF_DUMMYS BY 1 DO
	MessageHandler.MessageLine[i].MsgTypeEnum:=MsgDataTypeString;
	MessageHandler.MessageLine[i].Text:=CONCAT('Dummy_',DINT_TO_STRING(i));
	IF Dummy_test_Result[i] THEN
		MessageHandler.MessageLine[i].MsgString:='OK';
	ELSE
		MessageHandler.MessageLine[i].MsgString:='NOK';
	END_IF
END_FOR


MessageHandler(
	Prio:=2, 								(*1=highest, .. , 4=lowest*)
	Btn1Addr:=ADR(MsgOk),						(*Address of Button1 , if Zero then Button is unvisible*)
	Btn2Addr:=0,						(*Address of Button2 , if Zero then Button is unvisible*)
	sVisu:=Visu.Message);
END_ACTION

ACTION Dummy_Test_Nok__exit:
MsgOk := FALSE;
END_ACTION

ACTION Dummy_Test_ok__entry:
MessageHandler.ClearMessageLines(sVisu:=Visu.Message);
END_ACTION

ACTION Dummy_Test_ok__action:
MessageHandler.Msg.ID:='PM54';
MessageHandler.Msg.Name:='DummyTest';
MessageHandler.Msg.Text:=' Dummy Pruefung OK, Ergebnis aller Teile OK ';
MessageHandler.Msg.Color:=Color.green;
MessageHandler.Msg.Station:=1;


MessageHandler(
	Prio:=2, 								(*1=highest, .. , 4=lowest*)
	Btn1Addr:=ADR(MsgOk),						(*Address of Button1 , if Zero then Button is unvisible*)
	Btn2Addr:=0,						(*Address of Button2 , if Zero then Button is unvisible*)
	sVisu:=Visu.Message);
END_ACTION

ACTION Dummy_Test_ok__exit:
MessageHandler.ClearMessageLines(sVisu:=Visu.Message);
MsgOk:=FALSE;
END_ACTION

ACTION SeqEnd_action:
IF 	State=STATE_RUN THEN
	SFCTime:=TIME_TO_DINT(TIME()-SFCTimeStart);
	State:=STATE_OK;
END_IF


IF 	NOT Start THEN
	State:=STATE_WAIT;
END_IF

StartErlaubt93pol:=TRUE;
END_ACTION

TRANSITION 160pol:
gTypeCode=322
END_TRANSITION

TRANSITION Empty:
ST08_CallPRGs.PosIdxHelp = 0
END_TRANSITION

TRANSITION #StateOK:
Robot01.State=STATE_OK

AND gTipImp
END_TRANSITION

TRANSITION 93_102pol:
(gTypeCode=312 OR			(*93pol*)
gTypeCode=499)	(*102pol*)
END_TRANSITION

TRANSITION Kamera_betriebsbereit:
(NOT ST02_DT_95_A1.b_kamera_aktiv (*Kamera Farberkennung*)
OR
NOT ST02_DT_95_A1.sm_kamera_nicht_bb) 	 (*Kamera Farberkennung*)
AND
(NOT ST02_DT_95_A2.sm_kamera_nicht_bb
OR
NOT ST02_DT_95_A2.Activated)
END_TRANSITION

TRANSITION DrehtellerLeer:
gTableEmpty=TRUE
END_TRANSITION

TRANSITION End_Test:
ST02_Main.LoopCounter >= 6
END_TRANSITION

TRANSITION OK_:
Dummy_ResOK=TRUE
END_TRANSITION

TRANSITION Reset_Dummytest:
MP.ST02.DummyPruefung_93pol = FALSE
END_TRANSITION

TRANSITION Reset_Dummytest:
MP.ST02.DummyPruefung_93pol = FALSE
END_TRANSITION

TRANSITION CheckState:
ST03_160pol_Zufuehrung.State = STATE_RUN
END_TRANSITION

TRANSITION DummyReady:
ST03_160pol_Zufuehrung.State <> STATE_RUN
END_TRANSITION

TRANSITION #StateOK:
Robot01.State=STATE_OK

AND gTipImp
END_TRANSITION

TRANSITION StateOk:
ST08_Process.State=STATE_OK
END_TRANSITION

TRANSITION StateWait:
ST08_Process.State=STATE_Wait
END_TRANSITION

TRANSITION Pal_OK:
ST08_Process.Pal_Ready=TRUE
END_TRANSITION

TRANSITION #StateOK:
Robot01.State=STATE_OK

AND gTipImp
END_TRANSITION

TRANSITION StateOk:
ST08_Process.State=STATE_OK OR ST08_Process.State=STATE_Wait
END_TRANSITION

TRANSITION Pal_OK:
ST08_Process.Pal_Ready=TRUE
END_TRANSITION

TRANSITION StateOK:
Robot01.State=STATE_OK
END_TRANSITION

TRANSITION #StateOK:
Robot01.State=STATE_OK

AND gTipImp
END_TRANSITION

TRANSITION StateRun:
ST08_Process.State=STATE_Run
END_TRANSITION

TRANSITION completed:
LoopCounter >= MAX_NO_OF_DUMMYS
END_TRANSITION

TRANSITION Ok:
Dummy_ResOK=TRUE
END_TRANSITION
END_PROGRAM

(* POU Stations/ST_08_Palettierer/ST_08_Programs/ST08_CallPRGs, ST *)
PROGRAM ST08_CallPRGs
VAR
	Delay      				: TON;
 	PosIdxHelpCopy 			: DINT;

	FB_ReadXmlLineConf		: FB_ReadXmlLine;
	sDescription			: STRING;
END_VAR
VAR_INPUT
 	PosIdxHelp : DINT;
END_VAR
IF 	ST02_HomePosition.State = STATE_RUN THEN
	ListHomeNOK(InstName:='ST02 ',Description:=sDescription);
END_IF
FB_ReadXmlLineConf(
	Prefix:= 'CONFIG',
	ID:= 'ST08',
	File:= 'CONFIG.xml',
	Text=> sDescription );

(*===================================================================*)
IF	PosIdxHelp<>PosIdxHelpCopy THEN
	PosIdxHelp:=PosIdxHelp - (PosIdxHelp MOD TD.PartsInRoboGripper);
	PosIdx:=PosIdxHelp+TD.PartsInRoboGripper;
	PosIdxHelpCopy:=PosIdxHelp;
ELSE
	PosIdxHelp:=PosIdx-TD.PartsInRoboGripper;
END_IF

(* Band Einlauf*)
IF 	ModeSelect.Mode>MODE_MANUAL THEN
	IF 	ST08_Depalletizing.ConveyorOn THEN
		ST08_169_K1.SetSignalHigh:=TRUE;
	ELSIF
		NOT ST08_Depalletizing.ConveyorOn THEN
    	ST08_169_K1.SetSignalLow:=TRUE;
	ELSE
	    ST08_169_K1.Reset:=TRUE;
	END_IF
END_IF

(* Band Hubquer*)
IF 	ModeSelect.Mode>MODE_MANUAL THEN
	IF 	ST08_Process.ConveyorHQE THEN
		ST08_170_K1.SetSignalHigh:=TRUE;
		ST08_170_K2.SetSignalHigh:=TRUE;
  	ELSIF
		NOT ST08_Process.ConveyorHQE THEN
    	ST08_170_K1.SetSignalLow:=TRUE;
    	ST08_170_K2.SetSignalLow:=TRUE;
	ELSE
		ST08_170_K1.Reset:=TRUE;
		ST08_170_K2.Reset:=TRUE;
	END_IF
END_IF

(* Band Einlauf*)

IF ModeSelect.Mode>MODE_MANUAL THEN
	IF 	ST08_Process.ConveyorOut OR ST08_Palletizing.ConveyorOn THEN
		ST08_169_K2.SetSignalHigh:=TRUE;
  	ELSIF
		ST08_Process.ConveyorOut= FALSE AND
		NOT ST08_Palletizing.ConveyorOn THEN
    	ST08_169_K2.SetSignalLow:=TRUE;
	ELSE
		ST08_169_K2.Reset:=TRUE;
	END_IF
END_IF

Delay(IN:=NOT ST08_409_B55_5.BitInToCheck,PT:=T#2000ms);

IF (ModeSelect.Mode=MODE_AUTO_RUN OR
	ModeSelect.Mode=MODE_STEP_RUN OR
  	ModeSelect.Mode=MODE_SPECIAL) AND
	Delay.Q THEN
	ProcessMessage01:='1IM5';(*... ST08 Auslaufband voll, bitte volle Blister entnehmen!*)
END_IF

(*Wenn die Anzahl Blister im Aufstapler gelöscht wird, dann muss nicht mehr aufgestapelt werden.*)
IF MP.ST08.NoOfBlisterInStackerOut=0 THEN
	ST08_Palletizing.MoveOut:=FALSE;
END_IF
END_PROGRAM

(* POU Stations/ST_02_RT_Tampondrucker/ST02_SFCs/ST02_HomePosition, SFC *)
PROGRAM ST02_HomePosition

VAR_OUTPUT
	SFCCurrentPOU		: STRING:='ST02_HomePosition';
	SFCCurrentStep		: STRING:='';
	SFCTime				: DINT;
	State   			: StateObject	:= STATE_WAIT;
	Result  			: StateResult;
END_VAR
VAR_INPUT
	Start				: BOOL;
END_VAR
VAR
	MsgOK				: BOOL;
	MsgCancel			: BOOL;
	SFCRun				: BOOL;
	SFCTimeStart		: TIME;
	(* Userdefinded area *)

END_VAR
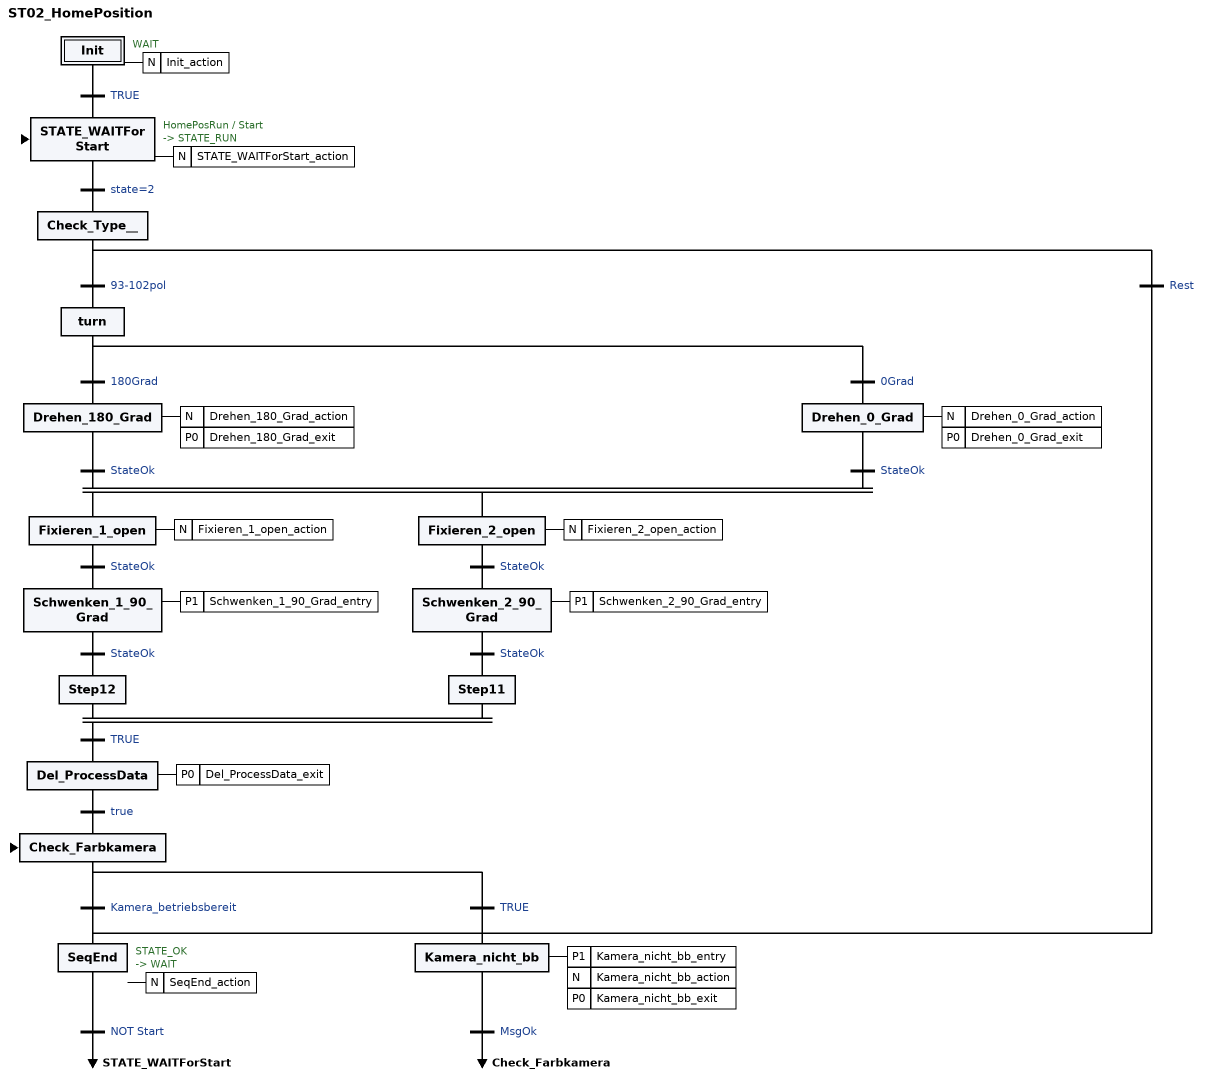
INITIAL_STEP Init: (* WAIT *)
	Init_action(N);
END_STEP
TRANSITION FROM Init TO STATE_WAITForStart := TRUE;
END_TRANSITION
STEP STATE_WAITForStart: (* HomePosRun / Start / -> STATE_RUN *)
	STATE_WAITForStart_action(N);
END_STEP
TRANSITION FROM STATE_WAITForStart TO Check_Type__ := state=2;
END_TRANSITION
STEP Check_Type__:
END_STEP
TRANSITION FROM Check_Type__ TO turn := 93-102pol;
END_TRANSITION
TRANSITION FROM Check_Type__ TO SeqEnd := Rest;
END_TRANSITION
STEP turn:
END_STEP
TRANSITION FROM turn TO Drehen_180_Grad := 180Grad;
END_TRANSITION
TRANSITION FROM turn TO Drehen_0_Grad := 0Grad;
END_TRANSITION
STEP Drehen_180_Grad:
	Drehen_180_Grad_action(N);
	Drehen_180_Grad_exit(P0);
END_STEP
TRANSITION FROM Drehen_180_Grad TO (Fixieren_1_open, Fixieren_2_open) := StateOk;
END_TRANSITION
STEP Drehen_0_Grad:
	Drehen_0_Grad_action(N);
	Drehen_0_Grad_exit(P0);
END_STEP
TRANSITION FROM Drehen_0_Grad TO (Fixieren_1_open, Fixieren_2_open) := StateOk;
END_TRANSITION
STEP Fixieren_1_open:
	Fixieren_1_open_action(N);
END_STEP
TRANSITION FROM Fixieren_1_open TO Schwenken_1_90_Grad := StateOk;
END_TRANSITION
STEP Schwenken_1_90_Grad:
	Schwenken_1_90_Grad_entry(P1);
END_STEP
TRANSITION FROM Schwenken_1_90_Grad TO Step12 := StateOk;
END_TRANSITION
STEP Step12:
END_STEP
STEP Fixieren_2_open:
	Fixieren_2_open_action(N);
END_STEP
TRANSITION FROM Fixieren_2_open TO Schwenken_2_90_Grad := StateOk;
END_TRANSITION
STEP Schwenken_2_90_Grad:
	Schwenken_2_90_Grad_entry(P1);
END_STEP
TRANSITION FROM Schwenken_2_90_Grad TO Step11 := StateOk;
END_TRANSITION
STEP Step11:
END_STEP
TRANSITION FROM (Step12, Step11) TO Del_ProcessData := TRUE;
END_TRANSITION
STEP Del_ProcessData:
	Del_ProcessData_exit(P0);
END_STEP
TRANSITION FROM Del_ProcessData TO Check_Farbkamera := true;
END_TRANSITION
STEP Check_Farbkamera:
END_STEP
TRANSITION FROM Check_Farbkamera TO SeqEnd := Kamera_betriebsbereit;
END_TRANSITION
TRANSITION FROM Check_Farbkamera TO Kamera_nicht_bb := TRUE;
END_TRANSITION
STEP Kamera_nicht_bb:
	Kamera_nicht_bb_entry(P1);
	Kamera_nicht_bb_action(N);
	Kamera_nicht_bb_exit(P0);
END_STEP
TRANSITION FROM Kamera_nicht_bb TO Check_Farbkamera := MsgOk;
END_TRANSITION
STEP SeqEnd: (* STATE_OK / -> WAIT *)
	SeqEnd_action(N);
END_STEP
TRANSITION FROM SeqEnd TO STATE_WAITForStart := NOT Start;
END_TRANSITION

ACTION Init_action:
Start:=FALSE;
State:=STATE_WAIT;
END_ACTION

ACTION STATE_WAITForStart_action:
IF	Start THEN
	State:=STATE_RUN;
	Result:=RESULT_NON;
	SFCTimeStart:=TIME();
ELSE
	;
END_IF
END_ACTION

ACTION Drehen_180_Grad_action:
ST02_62_Y6.MoveWork:=TRUE;
END_ACTION

ACTION Drehen_180_Grad_exit:
MP.ST02.TableData:=PushData(MP.ST02.TableData);


MP.ST02.TableData[1].ProcessData.	Result:=0;	(*   0 = Teil noch nicht bearbeitet *)
											(*   1 =  Oberseite OK*)
											(*  11 = Oberseite und Unterseite OK*)
											(*  99 = Teil ist NOK	*)
END_ACTION

ACTION Drehen_0_Grad_action:
ST02_62_Y6.MoveInit:=TRUE;
END_ACTION

ACTION Drehen_0_Grad_exit:
MP.ST02.TableData:=PushData(MP.ST02.TableData);


MP.ST02.TableData[1].ProcessData.	Result:=0;	(*   0 = Teil noch nicht bearbeitet *)
											(*   1 =  Oberseite OK*)
											(*  11 = Oberseite und Unterseite OK*)
											(*  99 = Teil ist NOK	*)
END_ACTION

ACTION Fixieren_1_open_action:
ST02_62_Y17.MoveInit:=TRUE;
END_ACTION

ACTION Schwenken_1_90_Grad_entry:
(*auf 180 Grad*)
ST02_Schwenkarm[1].b_90_grad:=TRUE;
END_ACTION

ACTION Fixieren_2_open_action:
ST02_62_Y18.MoveInit:=TRUE;
END_ACTION

ACTION Schwenken_2_90_Grad_entry:
(*auf 180 Grad*)
ST02_Schwenkarm[2].b_90_grad:=TRUE;
END_ACTION

ACTION Del_ProcessData_exit:
IF	NOT ST02_DT_65B11.BitInToCheck THEN
	MP.ST02.TableData[2].ProcessData.Result:=99;
END_IF
MP.ST02.TableData[2].ProcessData.Part:= NOT ST02_DT_65B11.BitInToCheck; 		 (* Tampondrucker Nest 1 leer *)

IF	NOT ST02_DT_65B21.BitInToCheck THEN
	MP.ST02.TableData[1].ProcessData.Result:=99;
END_IF
MP.ST02.TableData[1].ProcessData.Part:= NOT ST02_DT_65B21.BitInToCheck; 		 (* Tampondrucker Nest 2 leer *)
END_ACTION

ACTION Kamera_nicht_bb_entry:
MessageHandler.ClearMessageLines(sVisu:=Visu.Message);
END_ACTION

ACTION Kamera_nicht_bb_action:
MessageHandler.Msg.Name:='cHECK cAMERA';
MessageHandler.Msg.Text:='Sesopart Kamera ist nicht betriebsbereit';
MessageHandler.Msg.Color:=Color.red;
MessageHandler.Msg.Station:=1;


MessageHandler(
	Prio:=2, 							(*1=highest, .. , 4=lowest*)
	Btn1Addr:=ADR(MsgOk),			(*Address of Button1 , if Zero then Button is unvisible*)
	Btn2Addr:=,						(*Address of Button2 , if Zero then Button is unvisible*)
	sVisu:=Visu.Message);
END_ACTION

ACTION Kamera_nicht_bb_exit:
MsgOk:=FALSE;
MsgCancel:=FALSE;
ST02_DT_95_A1.b_quitt:=TRUE;
END_ACTION

ACTION SeqEnd_action:
IF 	State=STATE_RUN THEN
	SFCTime:=TIME_TO_DINT(TIME()-SFCTimeStart);
	State:=STATE_OK;
END_IF

IF 	NOT Start THEN
	State:=STATE_WAIT;
END_IF
END_ACTION

TRANSITION 93-102pol:
TRUE
END_TRANSITION

TRANSITION 180Grad:
ST02_DT_62_B91.ValveSensor				(* Tisch  180 Grad*)
END_TRANSITION

TRANSITION StateOk:
ST02_62_Y6.State=STATE_OK
END_TRANSITION

TRANSITION 0Grad:
TRUE
(*ST02_DT_62_B81.ValveSensor 	(* Tisch  0 Grad*)*)
END_TRANSITION

TRANSITION StateOk:
ST02_62_Y6.State=STATE_OK
END_TRANSITION

TRANSITION StateOk:
ST02_62_Y17.State=STATE_OK
AND
gTipImp
END_TRANSITION

TRANSITION StateOk:
NOT ST02_Schwenkarm[1].b_90_grad AND
ST02_Schwenkarm[1].b_done
END_TRANSITION

TRANSITION StateOk:
ST02_62_Y18.State=STATE_OK
AND
gTipImp
END_TRANSITION

TRANSITION StateOk:
NOT ST02_Schwenkarm[2].b_90_grad AND
ST02_Schwenkarm[2].b_done
END_TRANSITION

TRANSITION Kamera_betriebsbereit:
(NOT ST02_DT_95_A1.b_kamera_aktiv (*Kamera Farberkennung*)
OR
NOT ST02_DT_95_A1.sm_kamera_nicht_bb) 	 (*Kamera Farberkennung*)
OR
NOT NOT ST02_DT_95_A2.sm_kamera_nicht_bb
OR
NOT ST02_DT_95_A2.Activated
END_TRANSITION

TRANSITION Rest:
TRUE
END_TRANSITION
END_PROGRAM

(* POU Stations/ST_02_RT_Tampondrucker/ST02_PRGs/PushData, ST *)
FUNCTION PushData : ARRAY[1..NO_OF_NEST] OF sStationData
VAR_INPUT
	TableData				: ARRAY[1..NO_OF_NEST] OF sStationData;
END_VAR
VAR
	DummyNest				: sProcessData;
END_VAR
DummyNest:=TableData[NO_OF_NEST].ProcessData; 			(* Speichere letztes Array in DummyNest *)


TableData[2].ProcessData:=TableData[1].ProcessData;


TableData[1].ProcessData:=DummyNest;					(* letztes Array (DummyNest) auf 1. Array kopieren *)

PushData:=TableData;
END_FUNCTION

(* POU System/GeneralFunctions/ListHomeNOK, ST *)
PROGRAM ListHomeNOK
VAR_OUTPUT
	HomeNOKArray			: ARRAY[1..ARRAY_SIZE] OF STRING(100);
END_VAR
VAR_INPUT
	InstName					:	STRING(30);		(* Name of instance  *)
	Description				:	STRING(255);		(* Description  *)
	Clear							: BOOL;
END_VAR
VAR
	ArrayIdx					: DINT;
END_VAR
VAR CONSTANT
	ARRAY_SIZE				: DINT :=30;
END_VAR
IF ArrayIdx < ARRAY_SIZE THEN
	ArrayIdx:=ArrayIdx+1;
	HomeNOKArray[ArrayIdx]:=CONCAT(CONCAT(InstName,': '),Description);
END_IF

IF 	Clear THEN
	Clear:=FALSE;
	FOR ArrayIdx:=1 TO ARRAY_SIZE DO
		HomeNOKArray[ArrayIdx]:='';
	END_FOR
	ArrayIdx:=0;
END_IF
END_PROGRAM

(* POU Stations/ST_08_Palettierer/ST_08_SFCs/ST08_Depalletizing, SFC *)
PROGRAM ST08_Depalletizing

VAR_OUTPUT
	SFCCurrentPOU			:STRING:='ST08_Depalletizing';
	SFCCurrentStep			:STRING:='';
	FB_CurrentStepHistorie	:FB_CurrentStepHistorie;
	SFCTime					:DINT;
	State   				: StateObject	:= STATE_WAIT;
	Result  				: StateResult;
	ConveyorOn				:BOOL;
END_VAR
VAR_INPUT
	Start							:	BOOL;
END_VAR
VAR
	MsgOK				:BOOL;
	MsgCancel			:BOOL;
	SFCRun				:BOOL;
	SFCTimeStart		:TIME;
	Delay				:TON;
	Timeout				:TON;
	DelayOut  			:TON;
	Error				:ErrorStruct;
	MsgString      		:STRING;
	MsgID		      	:STRING(20);
	(* Userdefinded area *)

	LockDepalletizing		:BOOL;

END_VAR
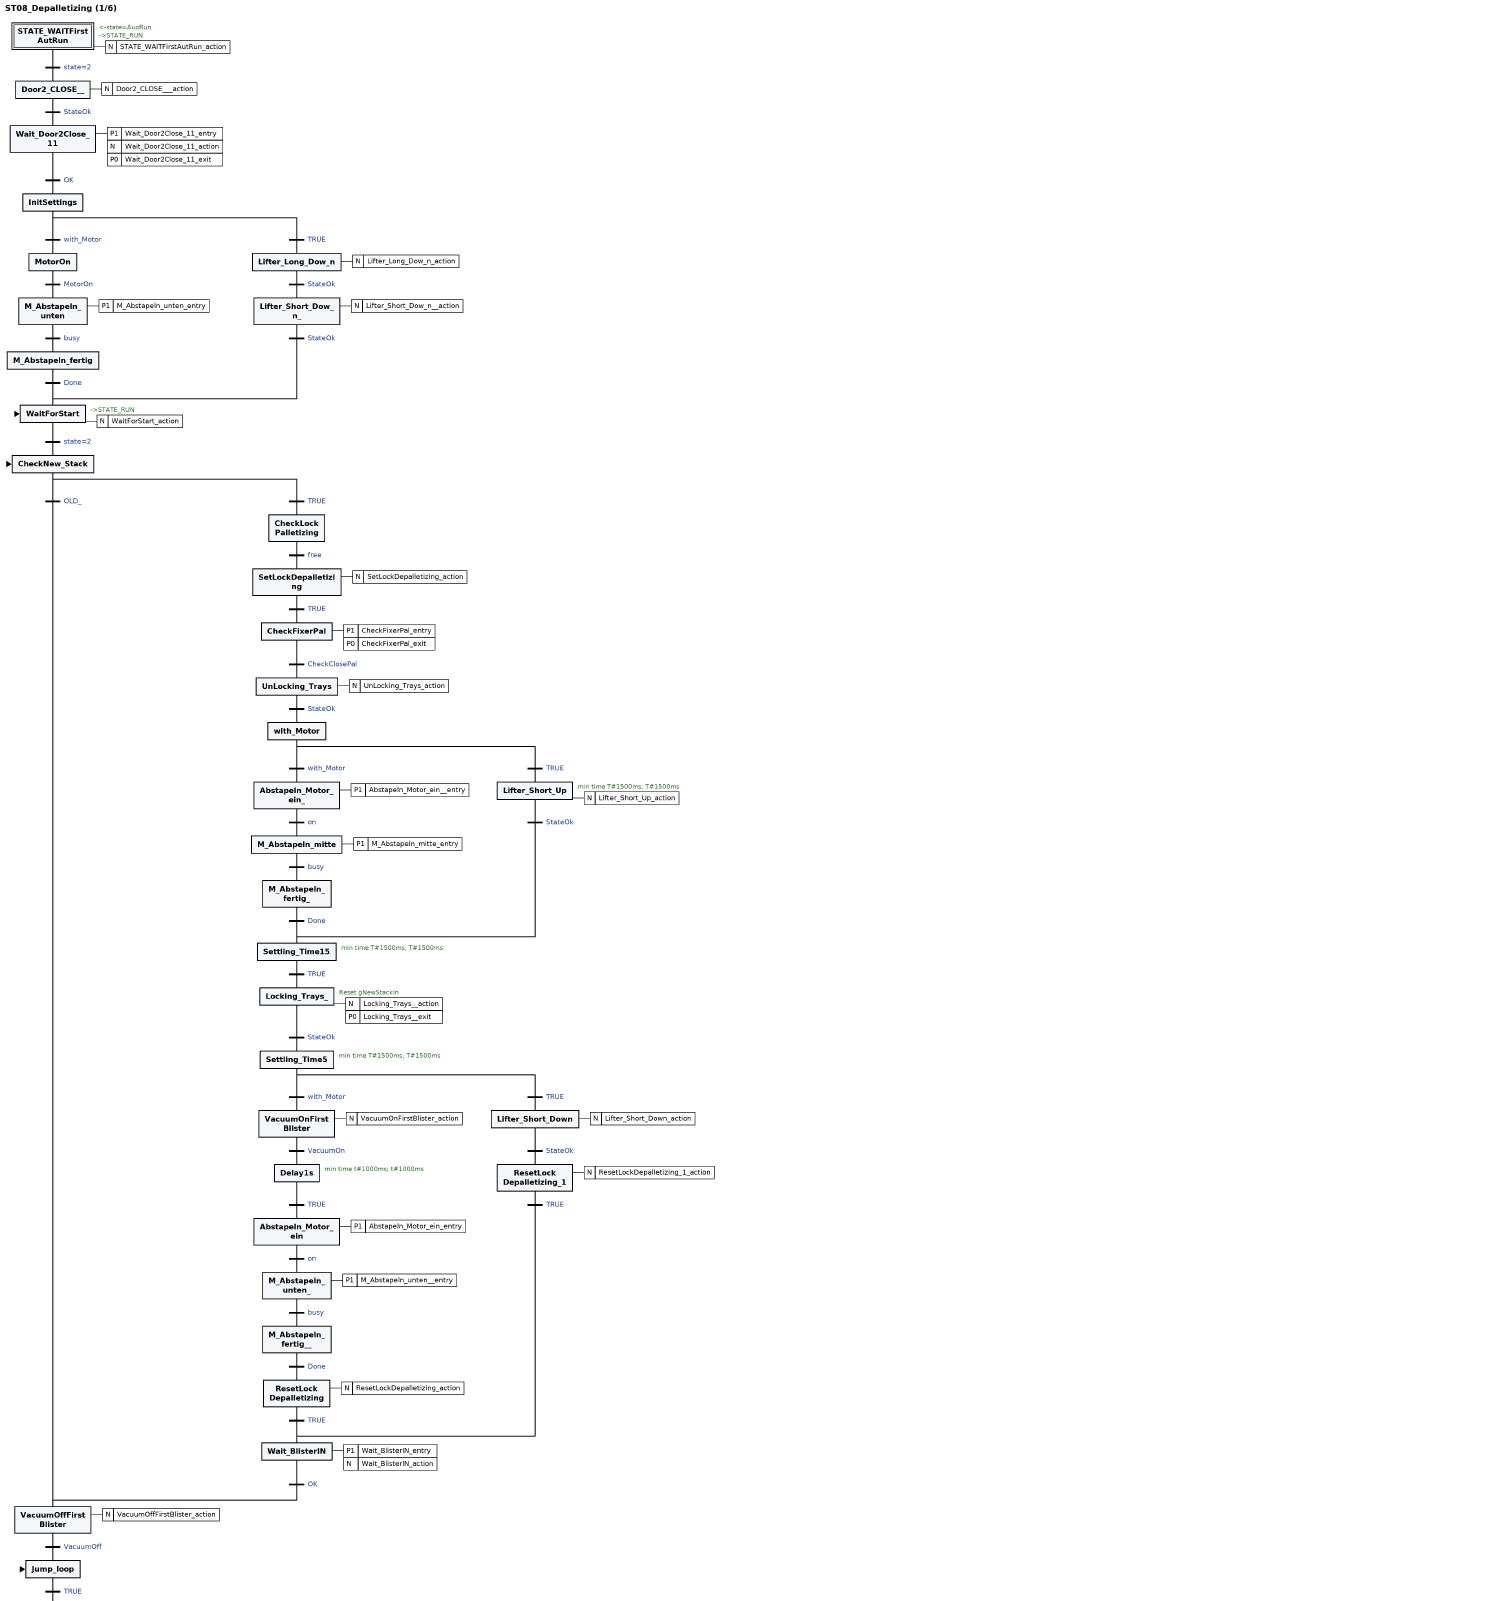
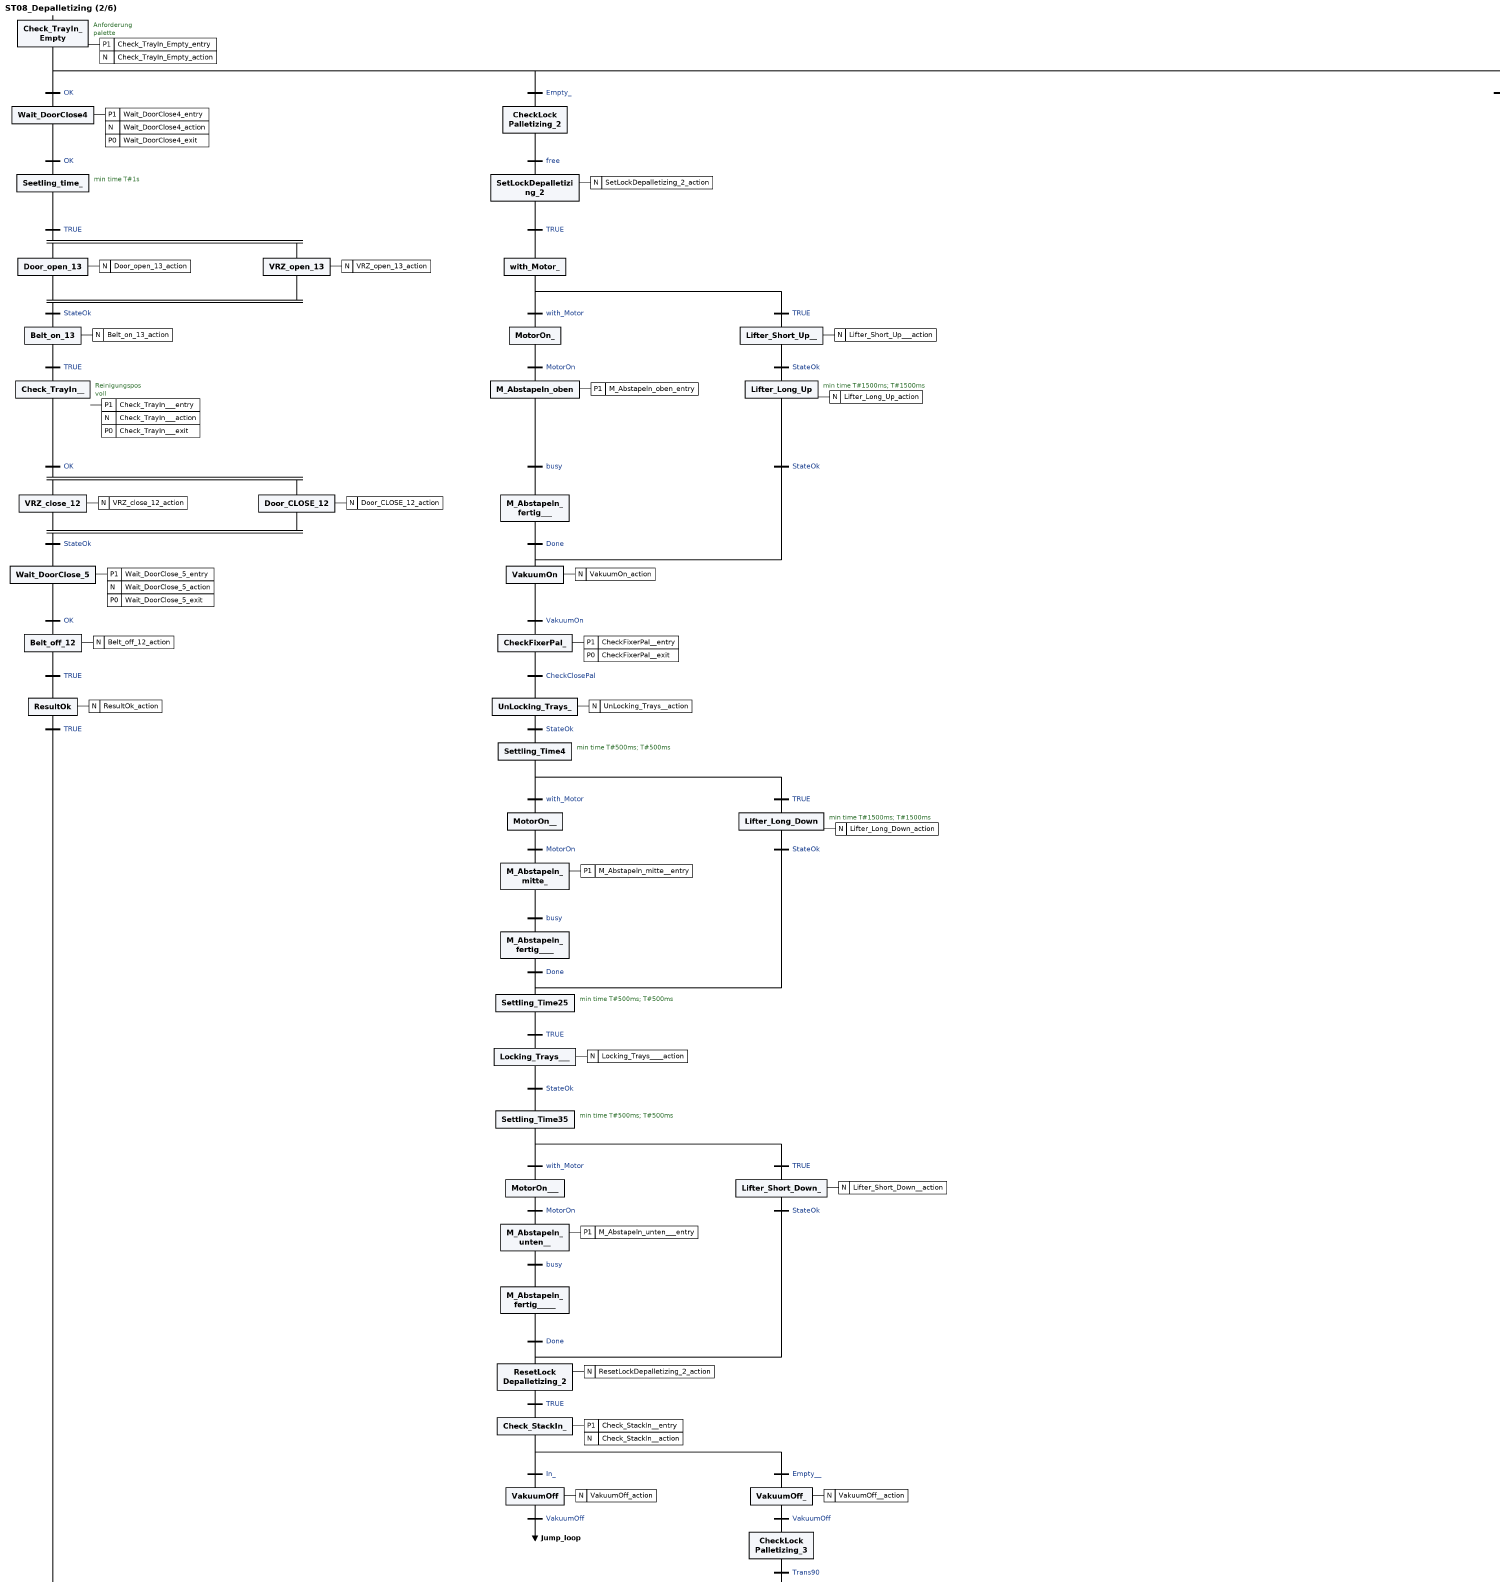
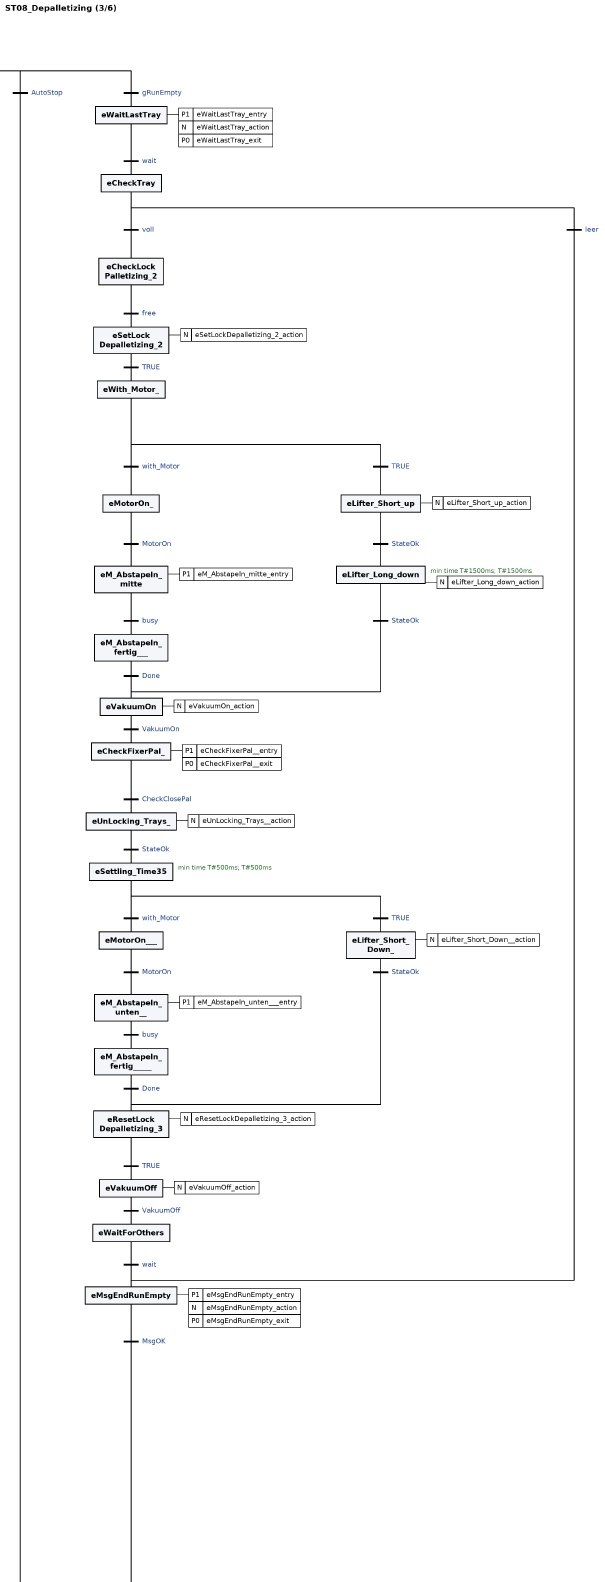
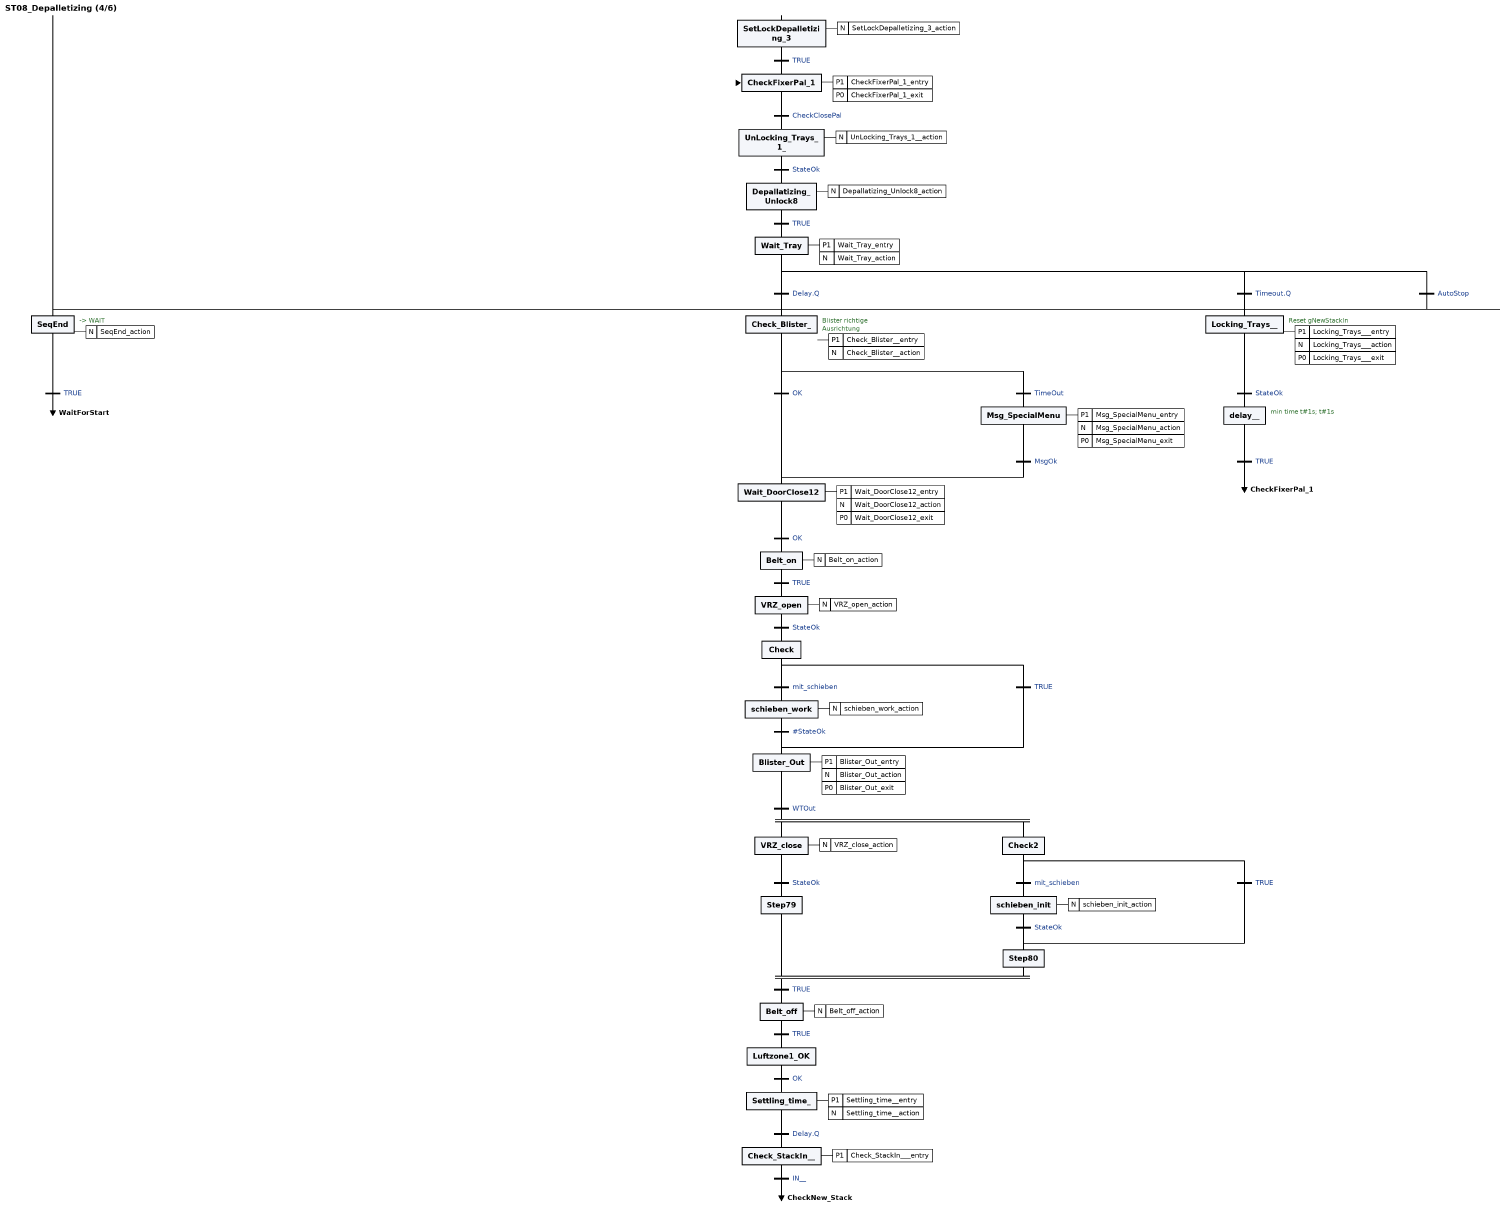
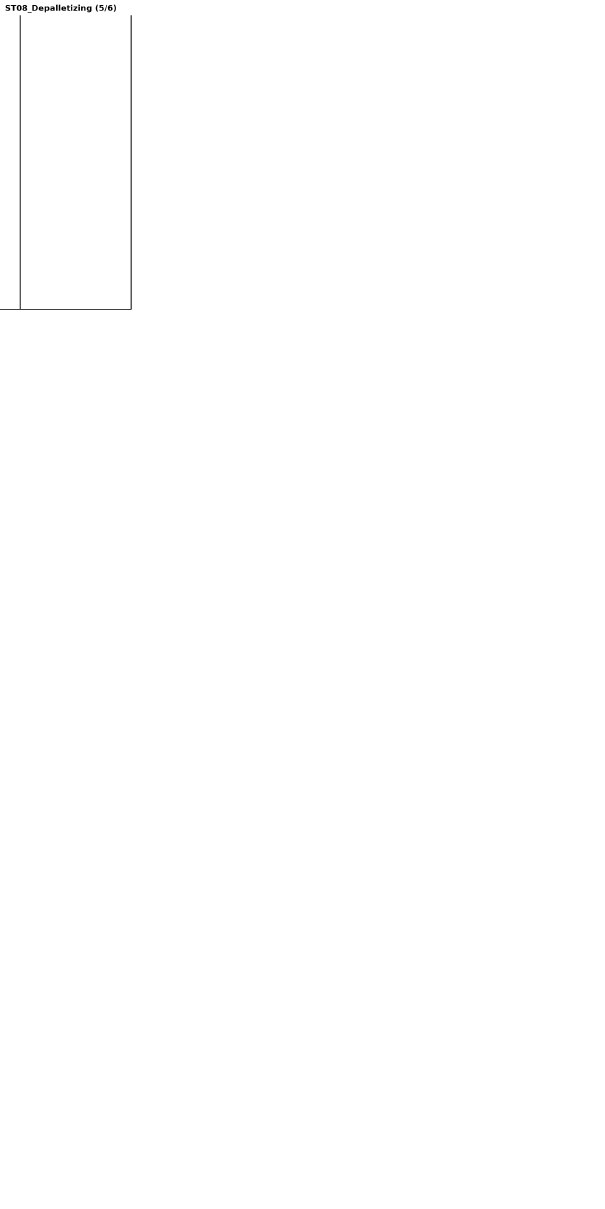
INITIAL_STEP STATE_WAITFirstAutRun: (* <-state=AuoRun / ->STATE_RUN *)
	STATE_WAITFirstAutRun_action(N);
END_STEP
TRANSITION FROM STATE_WAITFirstAutRun TO Door2_CLOSE__ := state=2;
END_TRANSITION
STEP Door2_CLOSE__:
	Door2_CLOSE___action(N);
END_STEP
TRANSITION FROM Door2_CLOSE__ TO Wait_Door2Close_11 := StateOk;
END_TRANSITION
STEP Wait_Door2Close_11:
	Wait_Door2Close_11_entry(P1);
	Wait_Door2Close_11_action(N);
	Wait_Door2Close_11_exit(P0);
END_STEP
TRANSITION FROM Wait_Door2Close_11 TO InitSettings := OK;
END_TRANSITION
STEP InitSettings:
END_STEP
TRANSITION FROM InitSettings TO MotorOn := with_Motor;
END_TRANSITION
TRANSITION FROM InitSettings TO Lifter_Long_Dow_n := TRUE;
END_TRANSITION
STEP MotorOn:
END_STEP
TRANSITION FROM MotorOn TO M_Abstapeln_unten := MotorOn;
END_TRANSITION
STEP M_Abstapeln_unten:
	M_Abstapeln_unten_entry(P1);
END_STEP
TRANSITION FROM M_Abstapeln_unten TO M_Abstapeln_fertig := busy;
END_TRANSITION
STEP M_Abstapeln_fertig:
END_STEP
TRANSITION FROM M_Abstapeln_fertig TO WaitForStart := Done;
END_TRANSITION
STEP Lifter_Long_Dow_n:
	Lifter_Long_Dow_n_action(N);
END_STEP
TRANSITION FROM Lifter_Long_Dow_n TO Lifter_Short_Dow_n_ := StateOk;
END_TRANSITION
STEP Lifter_Short_Dow_n_:
	Lifter_Short_Dow_n__action(N);
END_STEP
TRANSITION FROM Lifter_Short_Dow_n_ TO WaitForStart := StateOk;
END_TRANSITION
STEP WaitForStart: (* ->STATE_RUN *)
	WaitForStart_action(N);
END_STEP
TRANSITION FROM WaitForStart TO CheckNew_Stack := state=2;
END_TRANSITION
STEP CheckNew_Stack:
END_STEP
TRANSITION FROM CheckNew_Stack TO VacuumOffFirstBlister := OLD_;
END_TRANSITION
TRANSITION FROM CheckNew_Stack TO CheckLockPalletizing := TRUE;
END_TRANSITION
STEP CheckLockPalletizing:
END_STEP
TRANSITION FROM CheckLockPalletizing TO SetLockDepalletizing := free;
END_TRANSITION
STEP SetLockDepalletizing:
	SetLockDepalletizing_action(N);
END_STEP
TRANSITION FROM SetLockDepalletizing TO CheckFixerPal := TRUE;
END_TRANSITION
STEP CheckFixerPal:
	CheckFixerPal_entry(P1);
	CheckFixerPal_exit(P0);
END_STEP
TRANSITION FROM CheckFixerPal TO UnLocking_Trays := CheckClosePal;
END_TRANSITION
STEP UnLocking_Trays:
	UnLocking_Trays_action(N);
END_STEP
TRANSITION FROM UnLocking_Trays TO with_Motor := StateOk;
END_TRANSITION
STEP with_Motor:
END_STEP
TRANSITION FROM with_Motor TO Abstapeln_Motor_ein_ := with_Motor;
END_TRANSITION
TRANSITION FROM with_Motor TO Lifter_Short_Up := TRUE;
END_TRANSITION
STEP Abstapeln_Motor_ein_:
	Abstapeln_Motor_ein__entry(P1);
END_STEP
TRANSITION FROM Abstapeln_Motor_ein_ TO M_Abstapeln_mitte := on;
END_TRANSITION
STEP M_Abstapeln_mitte:
	M_Abstapeln_mitte_entry(P1);
END_STEP
TRANSITION FROM M_Abstapeln_mitte TO M_Abstapeln_fertig_ := busy;
END_TRANSITION
STEP M_Abstapeln_fertig_:
END_STEP
TRANSITION FROM M_Abstapeln_fertig_ TO Settling_Time15 := Done;
END_TRANSITION
STEP Lifter_Short_Up: (* min time T#1500ms; T#1500ms *)
	Lifter_Short_Up_action(N);
END_STEP
TRANSITION FROM Lifter_Short_Up TO Settling_Time15 := StateOk;
END_TRANSITION
STEP Settling_Time15: (* min time T#1500ms; T#1500ms *)
END_STEP
TRANSITION FROM Settling_Time15 TO Locking_Trays_ := TRUE;
END_TRANSITION
STEP Locking_Trays_: (* Reset gNewStackIn *)
	Locking_Trays__action(N);
	Locking_Trays__exit(P0);
END_STEP
TRANSITION FROM Locking_Trays_ TO Settling_Time5 := StateOk;
END_TRANSITION
STEP Settling_Time5: (* min time T#1500ms; T#1500ms *)
END_STEP
TRANSITION FROM Settling_Time5 TO VacuumOnFirstBlister := with_Motor;
END_TRANSITION
TRANSITION FROM Settling_Time5 TO Lifter_Short_Down := TRUE;
END_TRANSITION
STEP VacuumOnFirstBlister:
	VacuumOnFirstBlister_action(N);
END_STEP
TRANSITION FROM VacuumOnFirstBlister TO Delay1s := VacuumOn;
END_TRANSITION
STEP Delay1s: (* min time t#1000ms; t#1000ms *)
END_STEP
TRANSITION FROM Delay1s TO Abstapeln_Motor_ein := TRUE;
END_TRANSITION
STEP Abstapeln_Motor_ein:
	Abstapeln_Motor_ein_entry(P1);
END_STEP
TRANSITION FROM Abstapeln_Motor_ein TO M_Abstapeln_unten_ := on;
END_TRANSITION
STEP M_Abstapeln_unten_:
	M_Abstapeln_unten__entry(P1);
END_STEP
TRANSITION FROM M_Abstapeln_unten_ TO M_Abstapeln_fertig__ := busy;
END_TRANSITION
STEP M_Abstapeln_fertig__:
END_STEP
TRANSITION FROM M_Abstapeln_fertig__ TO ResetLockDepalletizing := Done;
END_TRANSITION
STEP ResetLockDepalletizing:
	ResetLockDepalletizing_action(N);
END_STEP
TRANSITION FROM ResetLockDepalletizing TO Wait_BlisterIN := TRUE;
END_TRANSITION
STEP Lifter_Short_Down:
	Lifter_Short_Down_action(N);
END_STEP
TRANSITION FROM Lifter_Short_Down TO ResetLockDepalletizing_1 := StateOk;
END_TRANSITION
STEP ResetLockDepalletizing_1:
	ResetLockDepalletizing_1_action(N);
END_STEP
TRANSITION FROM ResetLockDepalletizing_1 TO Wait_BlisterIN := TRUE;
END_TRANSITION
STEP Wait_BlisterIN:
	Wait_BlisterIN_entry(P1);
	Wait_BlisterIN_action(N);
END_STEP
TRANSITION FROM Wait_BlisterIN TO VacuumOffFirstBlister := OK;
END_TRANSITION
STEP VacuumOffFirstBlister:
	VacuumOffFirstBlister_action(N);
END_STEP
TRANSITION FROM VacuumOffFirstBlister TO Jump_loop := VacuumOff;
END_TRANSITION
STEP Jump_loop:
END_STEP
TRANSITION FROM Jump_loop TO Check_TrayIn_Empty := TRUE;
END_TRANSITION
STEP Check_TrayIn_Empty: (* Anforderung / palette *)
	Check_TrayIn_Empty_entry(P1);
	Check_TrayIn_Empty_action(N);
END_STEP
TRANSITION FROM Check_TrayIn_Empty TO Wait_DoorClose4 := OK;
END_TRANSITION
TRANSITION FROM Check_TrayIn_Empty TO CheckLockPalletizing_2 := Empty_;
END_TRANSITION
TRANSITION FROM Check_TrayIn_Empty TO SeqEnd := AutoStop;
END_TRANSITION
TRANSITION FROM Check_TrayIn_Empty TO eWaitLastTray := gRunEmpty;
END_TRANSITION
STEP CheckLockPalletizing_2:
END_STEP
TRANSITION FROM CheckLockPalletizing_2 TO SetLockDepalletizing_2 := free;
END_TRANSITION
STEP SetLockDepalletizing_2:
	SetLockDepalletizing_2_action(N);
END_STEP
TRANSITION FROM SetLockDepalletizing_2 TO with_Motor_ := TRUE;
END_TRANSITION
STEP with_Motor_:
END_STEP
TRANSITION FROM with_Motor_ TO MotorOn_ := with_Motor;
END_TRANSITION
TRANSITION FROM with_Motor_ TO Lifter_Short_Up__ := TRUE;
END_TRANSITION
STEP MotorOn_:
END_STEP
TRANSITION FROM MotorOn_ TO M_Abstapeln_oben := MotorOn;
END_TRANSITION
STEP M_Abstapeln_oben:
	M_Abstapeln_oben_entry(P1);
END_STEP
TRANSITION FROM M_Abstapeln_oben TO M_Abstapeln_fertig___ := busy;
END_TRANSITION
STEP M_Abstapeln_fertig___:
END_STEP
TRANSITION FROM M_Abstapeln_fertig___ TO VakuumOn := Done;
END_TRANSITION
STEP Lifter_Short_Up__:
	Lifter_Short_Up___action(N);
END_STEP
TRANSITION FROM Lifter_Short_Up__ TO Lifter_Long_Up := StateOk;
END_TRANSITION
STEP Lifter_Long_Up: (* min time T#1500ms; T#1500ms *)
	Lifter_Long_Up_action(N);
END_STEP
TRANSITION FROM Lifter_Long_Up TO VakuumOn := StateOk;
END_TRANSITION
STEP VakuumOn:
	VakuumOn_action(N);
END_STEP
TRANSITION FROM VakuumOn TO CheckFixerPal_ := VakuumOn;
END_TRANSITION
STEP CheckFixerPal_:
	CheckFixerPal__entry(P1);
	CheckFixerPal__exit(P0);
END_STEP
TRANSITION FROM CheckFixerPal_ TO UnLocking_Trays_ := CheckClosePal;
END_TRANSITION
STEP UnLocking_Trays_:
	UnLocking_Trays__action(N);
END_STEP
TRANSITION FROM UnLocking_Trays_ TO Settling_Time4 := StateOk;
END_TRANSITION
STEP Settling_Time4: (* min time T#500ms; T#500ms *)
END_STEP
TRANSITION FROM Settling_Time4 TO MotorOn__ := with_Motor;
END_TRANSITION
TRANSITION FROM Settling_Time4 TO Lifter_Long_Down := TRUE;
END_TRANSITION
STEP MotorOn__:
END_STEP
TRANSITION FROM MotorOn__ TO M_Abstapeln_mitte_ := MotorOn;
END_TRANSITION
STEP M_Abstapeln_mitte_:
	M_Abstapeln_mitte__entry(P1);
END_STEP
TRANSITION FROM M_Abstapeln_mitte_ TO M_Abstapeln_fertig____ := busy;
END_TRANSITION
STEP M_Abstapeln_fertig____:
END_STEP
TRANSITION FROM M_Abstapeln_fertig____ TO Settling_Time25 := Done;
END_TRANSITION
STEP Lifter_Long_Down: (* min time T#1500ms; T#1500ms *)
	Lifter_Long_Down_action(N);
END_STEP
TRANSITION FROM Lifter_Long_Down TO Settling_Time25 := StateOk;
END_TRANSITION
STEP Settling_Time25: (* min time T#500ms; T#500ms *)
END_STEP
TRANSITION FROM Settling_Time25 TO Locking_Trays___ := TRUE;
END_TRANSITION
STEP Locking_Trays___:
	Locking_Trays____action(N);
END_STEP
TRANSITION FROM Locking_Trays___ TO Settling_Time35 := StateOk;
END_TRANSITION
STEP Settling_Time35: (* min time T#500ms; T#500ms *)
END_STEP
TRANSITION FROM Settling_Time35 TO MotorOn___ := with_Motor;
END_TRANSITION
TRANSITION FROM Settling_Time35 TO Lifter_Short_Down_ := TRUE;
END_TRANSITION
STEP MotorOn___:
END_STEP
TRANSITION FROM MotorOn___ TO M_Abstapeln_unten__ := MotorOn;
END_TRANSITION
STEP M_Abstapeln_unten__:
	M_Abstapeln_unten___entry(P1);
END_STEP
TRANSITION FROM M_Abstapeln_unten__ TO M_Abstapeln_fertig_____ := busy;
END_TRANSITION
STEP M_Abstapeln_fertig_____:
END_STEP
TRANSITION FROM M_Abstapeln_fertig_____ TO ResetLockDepalletizing_2 := Done;
END_TRANSITION
STEP Lifter_Short_Down_:
	Lifter_Short_Down__action(N);
END_STEP
TRANSITION FROM Lifter_Short_Down_ TO ResetLockDepalletizing_2 := StateOk;
END_TRANSITION
STEP ResetLockDepalletizing_2:
	ResetLockDepalletizing_2_action(N);
END_STEP
TRANSITION FROM ResetLockDepalletizing_2 TO Check_StackIn_ := TRUE;
END_TRANSITION
STEP Check_StackIn_:
	Check_StackIn__entry(P1);
	Check_StackIn__action(N);
END_STEP
TRANSITION FROM Check_StackIn_ TO VakuumOff := In_;
END_TRANSITION
TRANSITION FROM Check_StackIn_ TO VakuumOff_ := Empty__;
END_TRANSITION
STEP VakuumOff:
	VakuumOff_action(N);
END_STEP
TRANSITION FROM VakuumOff TO Jump_loop := VakuumOff;
END_TRANSITION
STEP VakuumOff_:
	VakuumOff__action(N);
END_STEP
TRANSITION FROM VakuumOff_ TO CheckLockPalletizing_3 := VakuumOff;
END_TRANSITION
STEP CheckLockPalletizing_3:
END_STEP
TRANSITION FROM CheckLockPalletizing_3 TO SetLockDepalletizing_3 := Trans90;
END_TRANSITION
STEP SetLockDepalletizing_3:
	SetLockDepalletizing_3_action(N);
END_STEP
TRANSITION FROM SetLockDepalletizing_3 TO CheckFixerPal_1 := TRUE;
END_TRANSITION
STEP CheckFixerPal_1:
	CheckFixerPal_1_entry(P1);
	CheckFixerPal_1_exit(P0);
END_STEP
TRANSITION FROM CheckFixerPal_1 TO UnLocking_Trays_1_ := CheckClosePal;
END_TRANSITION
STEP UnLocking_Trays_1_:
	UnLocking_Trays_1__action(N);
END_STEP
TRANSITION FROM UnLocking_Trays_1_ TO Depallatizing_Unlock8 := StateOk;
END_TRANSITION
STEP Depallatizing_Unlock8:
	Depallatizing_Unlock8_action(N);
END_STEP
TRANSITION FROM Depallatizing_Unlock8 TO Wait_Tray := TRUE;
END_TRANSITION
STEP Wait_Tray:
	Wait_Tray_entry(P1);
	Wait_Tray_action(N);
END_STEP
TRANSITION FROM Wait_Tray TO Check_Blister_ := Delay.Q;
END_TRANSITION
TRANSITION FROM Wait_Tray TO Locking_Trays__ := Timeout.Q;
END_TRANSITION
TRANSITION FROM Wait_Tray TO SeqEnd := AutoStop;
END_TRANSITION
STEP Locking_Trays__: (* Reset gNewStackIn *)
	Locking_Trays___entry(P1);
	Locking_Trays___action(N);
	Locking_Trays___exit(P0);
END_STEP
TRANSITION FROM Locking_Trays__ TO delay__ := StateOk;
END_TRANSITION
STEP delay__: (* min time t#1s; t#1s *)
END_STEP
TRANSITION FROM delay__ TO CheckFixerPal_1 := TRUE;
END_TRANSITION
STEP Check_Blister_: (* Blister richtige / Ausrichtung *)
	Check_Blister__entry(P1);
	Check_Blister__action(N);
END_STEP
TRANSITION FROM Check_Blister_ TO Wait_DoorClose12 := OK;
END_TRANSITION
TRANSITION FROM Check_Blister_ TO Msg_SpecialMenu := TimeOut;
END_TRANSITION
STEP Msg_SpecialMenu:
	Msg_SpecialMenu_entry(P1);
	Msg_SpecialMenu_action(N);
	Msg_SpecialMenu_exit(P0);
END_STEP
TRANSITION FROM Msg_SpecialMenu TO Wait_DoorClose12 := MsgOk;
END_TRANSITION
STEP Wait_DoorClose12:
	Wait_DoorClose12_entry(P1);
	Wait_DoorClose12_action(N);
	Wait_DoorClose12_exit(P0);
END_STEP
TRANSITION FROM Wait_DoorClose12 TO Belt_on := OK;
END_TRANSITION
STEP Belt_on:
	Belt_on_action(N);
END_STEP
TRANSITION FROM Belt_on TO VRZ_open := TRUE;
END_TRANSITION
STEP VRZ_open:
	VRZ_open_action(N);
END_STEP
TRANSITION FROM VRZ_open TO Check := StateOk;
END_TRANSITION
STEP Check:
END_STEP
TRANSITION FROM Check TO schieben_work := mit_schieben;
END_TRANSITION
TRANSITION FROM Check TO Blister_Out := TRUE;
END_TRANSITION
STEP schieben_work:
	schieben_work_action(N);
END_STEP
TRANSITION FROM schieben_work TO Blister_Out := #StateOk;
END_TRANSITION
STEP Blister_Out:
	Blister_Out_entry(P1);
	Blister_Out_action(N);
	Blister_Out_exit(P0);
END_STEP
TRANSITION FROM Blister_Out TO (VRZ_close, Check2) := WTOut;
END_TRANSITION
STEP VRZ_close:
	VRZ_close_action(N);
END_STEP
TRANSITION FROM VRZ_close TO Step79 := StateOk;
END_TRANSITION
STEP Step79:
END_STEP
STEP Check2:
END_STEP
TRANSITION FROM Check2 TO schieben_init := mit_schieben;
END_TRANSITION
TRANSITION FROM Check2 TO Step80 := TRUE;
END_TRANSITION
STEP schieben_init:
	schieben_init_action(N);
END_STEP
TRANSITION FROM schieben_init TO Step80 := StateOk;
END_TRANSITION
STEP Step80:
END_STEP
TRANSITION FROM (Step79, Step80) TO Belt_off := TRUE;
END_TRANSITION
STEP Belt_off:
	Belt_off_action(N);
END_STEP
TRANSITION FROM Belt_off TO Luftzone1_OK := TRUE;
END_TRANSITION
STEP Luftzone1_OK:
END_STEP
TRANSITION FROM Luftzone1_OK TO Settling_time_ := OK;
END_TRANSITION
STEP Settling_time_:
	Settling_time__entry(P1);
	Settling_time__action(N);
END_STEP
TRANSITION FROM Settling_time_ TO Check_StackIn__ := Delay.Q;
END_TRANSITION
STEP Check_StackIn__:
	Check_StackIn___entry(P1);
END_STEP
TRANSITION FROM Check_StackIn__ TO CheckNew_Stack := IN__;
END_TRANSITION
STEP Wait_DoorClose4:
	Wait_DoorClose4_entry(P1);
	Wait_DoorClose4_action(N);
	Wait_DoorClose4_exit(P0);
END_STEP
TRANSITION FROM Wait_DoorClose4 TO Seetling_time_ := OK;
END_TRANSITION
STEP Seetling_time_: (* min time T#1s *)
END_STEP
TRANSITION FROM Seetling_time_ TO (Door_open_13, VRZ_open_13) := TRUE;
END_TRANSITION
STEP Door_open_13:
	Door_open_13_action(N);
END_STEP
STEP VRZ_open_13:
	VRZ_open_13_action(N);
END_STEP
TRANSITION FROM (Door_open_13, VRZ_open_13) TO Belt_on_13 := StateOk;
END_TRANSITION
STEP Belt_on_13:
	Belt_on_13_action(N);
END_STEP
TRANSITION FROM Belt_on_13 TO Check_TrayIn__ := TRUE;
END_TRANSITION
STEP Check_TrayIn__: (* Reinigungspos / voll *)
	Check_TrayIn___entry(P1);
	Check_TrayIn___action(N);
	Check_TrayIn___exit(P0);
END_STEP
TRANSITION FROM Check_TrayIn__ TO (VRZ_close_12, Door_CLOSE_12) := OK;
END_TRANSITION
STEP VRZ_close_12:
	VRZ_close_12_action(N);
END_STEP
STEP Door_CLOSE_12:
	Door_CLOSE_12_action(N);
END_STEP
TRANSITION FROM (VRZ_close_12, Door_CLOSE_12) TO Wait_DoorClose_5 := StateOk;
END_TRANSITION
STEP Wait_DoorClose_5:
	Wait_DoorClose_5_entry(P1);
	Wait_DoorClose_5_action(N);
	Wait_DoorClose_5_exit(P0);
END_STEP
TRANSITION FROM Wait_DoorClose_5 TO Belt_off_12 := OK;
END_TRANSITION
STEP Belt_off_12:
	Belt_off_12_action(N);
END_STEP
TRANSITION FROM Belt_off_12 TO ResultOk := TRUE;
END_TRANSITION
STEP ResultOk:
	ResultOk_action(N);
END_STEP
TRANSITION FROM ResultOk TO SeqEnd := TRUE;
END_TRANSITION
STEP eWaitLastTray:
	eWaitLastTray_entry(P1);
	eWaitLastTray_action(N);
	eWaitLastTray_exit(P0);
END_STEP
TRANSITION FROM eWaitLastTray TO eCheckTray := wait;
END_TRANSITION
STEP eCheckTray:
END_STEP
TRANSITION FROM eCheckTray TO eCheckLockPalletizing_2 := voll;
END_TRANSITION
TRANSITION FROM eCheckTray TO eMsgEndRunEmpty := leer;
END_TRANSITION
STEP eCheckLockPalletizing_2:
END_STEP
TRANSITION FROM eCheckLockPalletizing_2 TO eSetLockDepalletizing_2 := free;
END_TRANSITION
STEP eSetLockDepalletizing_2:
	eSetLockDepalletizing_2_action(N);
END_STEP
TRANSITION FROM eSetLockDepalletizing_2 TO eWith_Motor_ := TRUE;
END_TRANSITION
STEP eWith_Motor_:
END_STEP
TRANSITION FROM eWith_Motor_ TO eMotorOn_ := with_Motor;
END_TRANSITION
TRANSITION FROM eWith_Motor_ TO eLifter_Short_up := TRUE;
END_TRANSITION
STEP eMotorOn_:
END_STEP
TRANSITION FROM eMotorOn_ TO eM_Abstapeln_mitte := MotorOn;
END_TRANSITION
STEP eM_Abstapeln_mitte:
	eM_Abstapeln_mitte_entry(P1);
END_STEP
TRANSITION FROM eM_Abstapeln_mitte TO eM_Abstapeln_fertig___ := busy;
END_TRANSITION
STEP eM_Abstapeln_fertig___:
END_STEP
TRANSITION FROM eM_Abstapeln_fertig___ TO eVakuumOn := Done;
END_TRANSITION
STEP eLifter_Short_up:
	eLifter_Short_up_action(N);
END_STEP
TRANSITION FROM eLifter_Short_up TO eLifter_Long_down := StateOk;
END_TRANSITION
STEP eLifter_Long_down: (* min time T#1500ms; T#1500ms *)
	eLifter_Long_down_action(N);
END_STEP
TRANSITION FROM eLifter_Long_down TO eVakuumOn := StateOk;
END_TRANSITION
STEP eVakuumOn:
	eVakuumOn_action(N);
END_STEP
TRANSITION FROM eVakuumOn TO eCheckFixerPal_ := VakuumOn;
END_TRANSITION
STEP eCheckFixerPal_:
	eCheckFixerPal__entry(P1);
	eCheckFixerPal__exit(P0);
END_STEP
TRANSITION FROM eCheckFixerPal_ TO eUnLocking_Trays_ := CheckClosePal;
END_TRANSITION
STEP eUnLocking_Trays_:
	eUnLocking_Trays__action(N);
END_STEP
TRANSITION FROM eUnLocking_Trays_ TO eSettling_Time35 := StateOk;
END_TRANSITION
STEP eSettling_Time35: (* min time T#500ms; T#500ms *)
END_STEP
TRANSITION FROM eSettling_Time35 TO eMotorOn___ := with_Motor;
END_TRANSITION
TRANSITION FROM eSettling_Time35 TO eLifter_Short_Down_ := TRUE;
END_TRANSITION
STEP eMotorOn___:
END_STEP
TRANSITION FROM eMotorOn___ TO eM_Abstapeln_unten__ := MotorOn;
END_TRANSITION
STEP eM_Abstapeln_unten__:
	eM_Abstapeln_unten___entry(P1);
END_STEP
TRANSITION FROM eM_Abstapeln_unten__ TO eM_Abstapeln_fertig_____ := busy;
END_TRANSITION
STEP eM_Abstapeln_fertig_____:
END_STEP
TRANSITION FROM eM_Abstapeln_fertig_____ TO eResetLockDepalletizing_3 := Done;
END_TRANSITION
STEP eLifter_Short_Down_:
	eLifter_Short_Down__action(N);
END_STEP
TRANSITION FROM eLifter_Short_Down_ TO eResetLockDepalletizing_3 := StateOk;
END_TRANSITION
STEP eResetLockDepalletizing_3:
	eResetLockDepalletizing_3_action(N);
END_STEP
TRANSITION FROM eResetLockDepalletizing_3 TO eVakuumOff := TRUE;
END_TRANSITION
STEP eVakuumOff:
	eVakuumOff_action(N);
END_STEP
TRANSITION FROM eVakuumOff TO eWaitForOthers := VakuumOff;
END_TRANSITION
STEP eWaitForOthers:
END_STEP
TRANSITION FROM eWaitForOthers TO eMsgEndRunEmpty := wait;
END_TRANSITION
STEP eMsgEndRunEmpty:
	eMsgEndRunEmpty_entry(P1);
	eMsgEndRunEmpty_action(N);
	eMsgEndRunEmpty_exit(P0);
END_STEP
TRANSITION FROM eMsgEndRunEmpty TO SeqEnd := MsgOK;
END_TRANSITION
STEP SeqEnd: (* -> WAIT *)
	SeqEnd_action(N);
END_STEP
TRANSITION FROM SeqEnd TO WaitForStart := TRUE;
END_TRANSITION

ACTION STATE_WAITFirstAutRun_action:
IF 	ModeSelect.Mode=MODE_AUTO_RUN OR
	ModeSelect.Mode=MODE_STEP_RUN OR
  	SpecialMode01.State=State_Run OR
	SpecialMode06.State=State_Run THEN
	State:=STATE_RUN;
	Result:=RESULT_NON;
ELSE
	State:=STATE_WAIT;
	SFCRun:=FALSE;
END_IF

LockDepalletizing := FALSE;

Start:=FALSE;
MsgOK:=FALSE;
MsgCancel:=FALSE;
ProcessMessage02:='EMPTY';
END_ACTION

ACTION Door2_CLOSE___action:
ST08_405_Y51_0.MoveInit:=TRUE; (*  Hubtüre 2 Einlauf Isokörper STN8 AST (Valve) *)
END_ACTION

ACTION Wait_Door2Close_11_entry:
ProcessMessage01:='';
END_ACTION

ACTION Wait_Door2Close_11_action:
ProcessMessage01:='1IM15';(*St.8 warte Türe 2 einlauf geschlossen*)
END_ACTION

ACTION Wait_Door2Close_11_exit:
ProcessMessage01:='';
END_ACTION

ACTION M_Abstapeln_unten_entry:
ST08_180_M1.MoveAbs:=TRUE;
ST08_180_M1.Vorgabe_Pos_Abs:=TD.PosAbstapeln[1].Pos;	(*1=unten, 2= mitte, 3=oben, 4=frei*)
ST08_180_M1.Vorgabe_Velo:=1750;
END_ACTION

ACTION Lifter_Long_Dow_n_action:
ST08_404_Y53_2.MoveInit:=TRUE;
END_ACTION

ACTION Lifter_Short_Dow_n__action:
ST08_404_Y53_0.MoveInit:=TRUE;
END_ACTION

ACTION WaitForStart_action:
 IF 	(	ModeSelect.Mode=MODE_AUTO_RUN OR 	ModeSelect.Mode=MODE_STEP_RUN   OR SpecialMode01.State=State_Run )

THEN
	State:=STATE_RUN;
	Result:=RESULT_NON;
	SFCTimeStart:=TIME();
(*ELSE*)
END_IF
END_ACTION

ACTION SetLockDepalletizing_action:
LockDepalletizing := TRUE;
END_ACTION

ACTION CheckFixerPal_entry:
ProcessMessage02:='2IM1';(*Abstapler wartet auf Aufstapler*)
END_ACTION

ACTION CheckFixerPal_exit:
ProcessMessage02:='';
END_ACTION

ACTION UnLocking_Trays_action:
ST08_405_Y53_4.MoveWork:=TRUE;
END_ACTION

ACTION Abstapeln_Motor_ein__entry:
ST08_180_M1.Vorgabe_Velo:=1750;
END_ACTION

ACTION M_Abstapeln_mitte_entry:
ST08_180_M1.MoveAbs:=TRUE;
ST08_180_M1.Vorgabe_Pos_Abs:=TD.PosAbstapeln[2].Pos;	(*1=unten, 2= mitte, 3=oben, 4=frei*)
END_ACTION

ACTION Lifter_Short_Up_action:
ST08_404_Y53_0.MoveWork:=TRUE;
END_ACTION

ACTION Locking_Trays__action:
ST08_405_Y53_4.MoveInit:=TRUE;
END_ACTION

ACTION Locking_Trays__exit:
gNewStackIn:=FALSE;
END_ACTION

ACTION VacuumOnFirstBlister_action:
ST08_403_Y50_6.MoveWork := TRUE;	(* Vakuum 1 Einlauf *)
ST08_403_Y50_7.MoveWork := TRUE;	(*Vakuum 2 Einlauf *)
END_ACTION

ACTION Abstapeln_Motor_ein_entry:
ST08_180_M1.Vorgabe_Velo:=1750;
END_ACTION

ACTION M_Abstapeln_unten__entry:
ST08_180_M1.MoveAbs:=TRUE;
ST08_180_M1.Vorgabe_Pos_Abs:=TD.PosAbstapeln[1].Pos;	(*1=unten, 2= mitte, 3=oben, 4=frei*)
END_ACTION

ACTION ResetLockDepalletizing_action:
LockDepalletizing := FALSE;
END_ACTION

ACTION Lifter_Short_Down_action:
ST08_404_Y53_0.MoveInit:=TRUE;
END_ACTION

ACTION ResetLockDepalletizing_1_action:
LockDepalletizing := FALSE;
END_ACTION

ACTION Wait_BlisterIN_entry:
Delay.IN:=FALSE;
Delay();
END_ACTION

ACTION Wait_BlisterIN_action:
Delay.IN:=TRUE;
Delay.PT:=T#3500ms;
Delay();
END_ACTION

ACTION VacuumOffFirstBlister_action:
ST08_403_Y50_6.MoveInit  := TRUE;	(* Vakuum 1 Einlauf *)
ST08_403_Y50_7.MoveInit  := TRUE;	(*Vakuum 2 Einlauf *)
END_ACTION

ACTION Check_TrayIn_Empty_entry:
Delay.IN:=FALSE;
Delay();
DelayOut.IN:=FALSE;
DelayOut();
END_ACTION

ACTION Check_TrayIn_Empty_action:
(*Mit Stapelmotor*)
IF MP.ST08.StapelMotor THEN
	Delay.IN:=
			ST08_404_B52_2.BitInToCheck AND		(*Traystapel in Ablageposition Isokörper*)
       		ABS(TD.PosAbstapeln[1].Pos -  ST08_180_M1.sPos.ist) < 0.1;
	Delay(PT:=T#500ms);
(*Ohne Stapelmotor*)
ELSE
	Delay.IN:=
			ST08_404_B52_2.BitInToCheck			(*Traystapel in Ablageposition Isokörper*)
      		AND ST08_404_Y53_0.InitPosition		(*Abstapelzylinder 1 Isokörper*)
      		AND ST08_404_Y53_2.InitPosition;	(*Abstapelzylinder 2 Isokörper*)
	Delay(PT:=T#500ms);
END_IF

DelayOut.IN:=
		ST08_404_Y52_0.InitPosition				(*Hub Bandstrecke AST*)
         AND ST08_406_B54_0.BitInToCheck		(* Tray in Zwischenp. Entnahme Isokörper (Bandende) *)
         AND NOT ST08_404_B52_2.BitInToCheck;	(*Traystapel in Ablageposition Isokörper*)
DelayOut(PT:=T#500ms);
END_ACTION

ACTION SetLockDepalletizing_2_action:
LockDepalletizing := TRUE;
END_ACTION

ACTION M_Abstapeln_oben_entry:
ST08_180_M1.MoveAbs:=TRUE;
ST08_180_M1.Vorgabe_Pos_Abs:=TD.PosAbstapeln[3].Pos;	(*1=unten, 2= mitte, 3=oben, 4=frei*)
END_ACTION

ACTION Lifter_Short_Up___action:
ST08_404_Y53_0.MoveWork:=TRUE;
END_ACTION

ACTION Lifter_Long_Up_action:
ST08_404_Y53_2.MoveWork:=TRUE;
END_ACTION

ACTION VakuumOn_action:
ST08_403_Y50_6.MoveWork := TRUE;
ST08_403_Y50_7.MoveWork := TRUE;
END_ACTION

ACTION CheckFixerPal__entry:
ProcessMessage02:='2IM1';(*'Abstapler wartet auf Aufstapler*)
END_ACTION

ACTION CheckFixerPal__exit:
ProcessMessage02:='';
END_ACTION

ACTION UnLocking_Trays__action:
ST08_405_Y53_4.MoveWork:=TRUE;
END_ACTION

ACTION M_Abstapeln_mitte__entry:
ST08_180_M1.MoveAbs:=TRUE;
ST08_180_M1.Vorgabe_Pos_Abs:=TD.PosAbstapeln[2].Pos;	(*1=unten, 2= mitte, 3=oben, 4=frei*)
END_ACTION

ACTION Lifter_Long_Down_action:
ST08_404_Y53_2.MoveInit:=TRUE;
END_ACTION

ACTION Locking_Trays____action:
ST08_405_Y53_4.MoveInit:=TRUE;
END_ACTION

ACTION M_Abstapeln_unten___entry:
ST08_180_M1.MoveAbs:=TRUE;
ST08_180_M1.Vorgabe_Pos_Abs:=TD.PosAbstapeln[1].Pos;	(*1=unten, 2= mitte, 3=oben, 4=frei*)
END_ACTION

ACTION Lifter_Short_Down__action:
ST08_404_Y53_0.MoveInit:=TRUE;
END_ACTION

